         $OUT[1167] = ($FLAG[330] OR $FLAG[331] OR NOT $FLAG[330] AND NOT $FLAG[331] AND NOT $FLAG[332]) AND NOT $TIMER_FLAG[9]
      ;ENDFOLD
      ;FOLD -- Warte Fraesen fertig oder Timeout -- ;%{SE}%MKUKATPVW %CVW_COM %VCOMMENT %P 2:-- Warte Fraesen fertig oder Timeout --, 3: VW_COMMENT
      ;ENDFOLD
      ;FOLD Schritt 107 = (F175 & F190 + F174 & F186 & !F287 + T7 + T9 + F325) & A4039  ;%{SE}%MKUKATPVW %CVW_SPS %VST_CON %P 2:Schritt 107 = (F175 & F190 + F174 & F186 & !F287 + T7 + T9 + F325) & A4039 , 3: ST_CON
         IF ($FLAG[175] AND $FLAG[190] OR $FLAG[174] AND $FLAG[186] AND NOT $FLAG[287] OR $TIMER_FLAG[7] OR $TIMER_FLAG[9] OR $FLAG[325]) AND $OUT[4039] THEN
            PREVSTEP = $APP_INT[5]
            $APP_INT[5] = 107
         ENDIF
      ;ENDFOLD
      ;FOLD Schritt 107 = (F174 & F188 & F287 + T7 + T9 + F325) & A4039  ;%{SE}%MKUKATPVW %CVW_SPS %VST_CON %P 2:Schritt 107 = (F174 & F188 & F287 + T7 + T9 + F325) & A4039 , 3: ST_CON
         IF ($FLAG[174] AND $FLAG[188] AND $FLAG[287] OR $TIMER_FLAG[7] OR $TIMER_FLAG[9] OR $FLAG[325]) AND $OUT[4039] THEN
            PREVSTEP = $APP_INT[5]
            $APP_INT[5] = 107
         ENDIF
      ;ENDFOLD
   ;ENDFOLD
   ;FOLD SCHRITT 107 -- STAT EZ3/SP3/KE3 -- ;%{P}%MKUKATPVW,%CSTEP,%VST_NR,%P 1:SCHRITT, 2:107, 3: STAT EZ3/SP3/KE3
      ;FOLD ;%{H}
         Case 107
      ;ENDFOLD
      ;FOLD t9 ( EIN ) = STOP ;%{SE}%MKUKATPVW %CVW_SPS %VTSTOP %P 2:t9 ( EIN ) = STOP, 3: TSTOP
         VW(#SET_TIME,TRUE,9,1,0)
      ;ENDFOLD
      ;FOLD -- EZ3/SP3/KE3 oeffnen -- ;%{SE}%MKUKATPVW %CVW_COM %VCOMMENT %P 2:-- EZ3/SP3/KE3 oeffnen --, 3: VW_COMMENT
      ;ENDFOLD
      ;FOLD A1039 = AUS ;%{SE}%MKUKATPVW %CVW_SPS %VBOASG %P 2:A1039 = AUS, 3: BOASG
         $OUT[1039] = FALSE
      ;ENDFOLD
      ;FOLD A1038 = AUS ;%{SE}%MKUKATPVW %CVW_SPS %VBOASG %P 2:A1038 = AUS, 3: BOASG
         $OUT[1038] = FALSE
      ;ENDFOLD
      ;FOLD A1037 = EIN ;%{SE}%MKUKATPVW %CVW_SPS %VBOASG %P 2:A1037 = EIN, 3: BOASG
         $OUT[1037] = TRUE
      ;ENDFOLD
      ;FOLD -- KF3 Ausblasen -- ;%{SE}%MKUKATPVW %CVW_COM %VCOMMENT %P 2:-- KF3 Ausblasen --, 3: VW_COMMENT
      ;ENDFOLD
      ;FOLD A1167 = F330 + F331 + F332 + !F330 & !F331 & !F332 ;%{SE}%MKUKATPVW %CVW_SPS %VBOASG %P 2:A1167 = F330 + F331 + F332 + !F330 & !F331 & !F332, 3: BOASG
         $OUT[1167] = $FLAG[330] OR $FLAG[331] OR $FLAG[332] OR NOT $FLAG[330] AND NOT $FLAG[331] AND NOT $FLAG[332]
      ;ENDFOLD
      ;FOLD -- KF Ausblasen Ausschaltverzoegerung starten -- ;%{SE}%MKUKATPVW %CVW_COM %VCOMMENT %P 2:-- KF Ausblasen Ausschaltverzoegerung starten --, 3: VW_COMMENT
      ;ENDFOLD
      ;FOLD F739 = EIN ;%{SE}%MKUKATPVW %CVW_SPS %VBOASG %P 2:F739 = EIN, 3: BOASG
         $FLAG[739] = TRUE
      ;ENDFOLD
      ;FOLD -- RSK Sammelstoerung -- ;%{SE}%MKUKATPVW %CVW_COM %VCOMMENT %P 2:-- RSK Sammelstoerung --, 3: VW_COMMENT
      ;ENDFOLD
      ;FOLD F329 = T7 + T9 + F325 ;%{SE}%MKUKATPVW %CVW_SPS %VBOASG %P 2:F329 = T7 + T9 + F325, 3: BOASG
         $FLAG[329] = $TIMER_FLAG[7] OR $TIMER_FLAG[9] OR $FLAG[325]
      ;ENDFOLD
      ;FOLD -- Hilfsflag Startfraesen -- ;%{SE}%MKUKATPVW %CVW_COM %VCOMMENT %P 2:-- Hilfsflag Startfraesen --, 3: VW_COMMENT
      ;ENDFOLD
      ;FOLD F188 = (F188 & F174 + F190 & F175) & F287 ;%{SE}%MKUKATPVW %CVW_SPS %VBOASG %P 2:F188 = (F188 & F174 + F190 & F175) & F287, 3: BOASG
         $FLAG[188] = ($FLAG[188] AND $FLAG[174] OR $FLAG[190] AND $FLAG[175]) AND $FLAG[287]
      ;ENDFOLD
      ;FOLD F190 = !F200 & F190 + F200 & F287 & F190 ;%{SE}%MKUKATPVW %CVW_SPS %VBOASG %P 2:F190 = !F200 & F190 + F200 & F287 & F190, 3: BOASG
         $FLAG[190] = NOT $FLAG[200] AND $FLAG[190] OR $FLAG[200] AND $FLAG[287] AND $FLAG[190]
      ;ENDFOLD
      ;FOLD F287 = F174 + F175 & F200 ;%{SE}%MKUKATPVW %CVW_SPS %VBOASG %P 2:F287 = F174 + F175 & F200, 3: BOASG
         $FLAG[287] = $FLAG[174] OR $FLAG[175] AND $FLAG[200]
      ;ENDFOLD
      ;FOLD -- Neues Fraesprogramm und Zaehler ruecksetzen -- ;%{SE}%MKUKATPVW %CVW_COM %VCOMMENT %P 2:-- Neues Fraesprogramm und Zaehler ruecksetzen --, 3: VW_COMMENT
      ;ENDFOLD
      ;FOLD F270 = F188 & F732 ;%{SE}%MKUKATPVW %CVW_SPS %VBOASG %P 2:F270 = F188 & F732, 3: BOASG
         $FLAG[270] = $FLAG[188] AND $FLAG[732]
      ;ENDFOLD
      ;FOLD bin9 ( F732 ) = 36 ;%{SE}%MKUKATPVW %CVW_SPS %VARIASG %P 2:bin9 ( F732 ) = 36, 3: ARIASG
         VW(#BINOUT,$FLAG[732],9,36)
      ;ENDFOLD
      ;FOLD i19 ( F270 ) = i45 ;%{SE}%MKUKATPVW %CVW_SPS %VARIASG %P 2:i19 ( F270 ) = i45, 3: ARIASG
         VW(#COUNTER,$FLAG[270],19,$COUNT_I[45])
      ;ENDFOLD
      ;FOLD -- Wiederholung beim Startfraesen -- ;%{SE}%MKUKATPVW %CVW_COM %VCOMMENT %P 2:-- Wiederholung beim Startfraesen --, 3: VW_COMMENT
      ;ENDFOLD
      ;FOLD Schritt 104 = E1037 & !E1038 & (F174 & !F188 + F175 & F200 & !F188) & !F325 & !F329 & A4039  ;%{SE}%MKUKATPVW %CVW_SPS %VST_CON %P 2:Schritt 104 = E1037 & !E1038 & (F174 & !F188 + F175 & F200 & !F188) & !F325 & !F329 & A4039 , 3: ST_CON
         IF $IN[1037] AND NOT $IN[1038] AND ($FLAG[174] AND NOT $FLAG[188] OR $FLAG[175] AND $FLAG[200] AND NOT $FLAG[188]) AND NOT $FLAG[325] AND NOT $FLAG[329] AND $OUT[4039] THEN
            PREVSTEP = $APP_INT[5]
            $APP_INT[5] = 104
         ENDIF
      ;ENDFOLD
      ;FOLD -- Weiter wenn Fraesen fertig -- ;%{SE}%MKUKATPVW %CVW_COM %VCOMMENT %P 2:-- Weiter wenn Fraesen fertig --, 3: VW_COMMENT
      ;ENDFOLD
      ;FOLD Schritt 108 = E1037 & !E1038 & (F175 & F190 & (!F200 + F188)+ F174 & F188 + F325 + F329) & A4039  ;%{SE}%MKUKATPVW %CVW_SPS %VST_CON %P 2:Schritt 108 = E1037 & !E1038 & (F175 & F190 & (!F200 + F188)+ F174 & F188 + F325 + F329) & A4039 , 3: ST_CON
         IF $IN[1037] AND NOT $IN[1038] AND ($FLAG[175] AND $FLAG[190] AND (NOT $FLAG[200] OR $FLAG[188]) OR $FLAG[174] AND $FLAG[188] OR $FLAG[325] OR $FLAG[329]) AND $OUT[4039] THEN
            PREVSTEP = $APP_INT[5]
            $APP_INT[5] = 108
         ENDIF
      ;ENDFOLD
   ;ENDFOLD
   ;FOLD SCHRITT 108 -- STAT EZ3/SP3/KE3 -- ;%{P}%MKUKATPVW,%CSTEP,%VST_NR,%P 1:SCHRITT, 2:108, 3: STAT EZ3/SP3/KE3
      ;FOLD ;%{H}
         Case 108
      ;ENDFOLD
      ;FOLD F270 = AUS ;%{SE}%MKUKATPVW %CVW_SPS %VBOASG %P 2:F270 = AUS, 3: BOASG
         $FLAG[270] = FALSE
      ;ENDFOLD
      ;FOLD F324 = AUS ;%{SE}%MKUKATPVW %CVW_SPS %VBOASG %P 2:F324 = AUS, 3: BOASG
         $FLAG[324] = FALSE
      ;ENDFOLD
      ;FOLD A1037 = AUS ;%{SE}%MKUKATPVW %CVW_SPS %VBOASG %P 2:A1037 = AUS, 3: BOASG
         $OUT[1037] = FALSE
      ;ENDFOLD
      ;FOLD -- KF3 abschalten -- ;%{SE}%MKUKATPVW %CVW_COM %VCOMMENT %P 2:-- KF3 abschalten --, 3: VW_COMMENT
      ;ENDFOLD
      ;FOLD A1154 = AUS ;%{SE}%MKUKATPVW %CVW_SPS %VBOASG %P 2:A1154 = AUS, 3: BOASG
         $OUT[1154] = FALSE
      ;ENDFOLD
      ;FOLD -- Ueberwachungszeit KF1 Versetzeinheit -- ;%{SE}%MKUKATPVW %CVW_COM %VCOMMENT %P 2:-- Ueberwachungszeit KF1 Versetzeinheit --, 3: VW_COMMENT
      ;ENDFOLD
      ;FOLD t8 ( EIN ) = -20[1/10Sek] ;%{SE}%MKUKATPVW %CVW_SPS %VTASG %P 2:t8 ( EIN ) = -20[1/10Sek], 3: TASG
         VW(#SET_TIME,TRUE,8,0,-20)
      ;ENDFOLD
      ;FOLD Schritt 109 = A4039  ;%{SE}%MKUKATPVW %CVW_SPS %VST_CON %P 2:Schritt 109 = A4039 , 3: ST_CON
         IF $OUT[4039] THEN
            PREVSTEP = $APP_INT[5]
            $APP_INT[5] = 109
         ENDIF
      ;ENDFOLD
   ;ENDFOLD
   ;FOLD SCHRITT 109 -- STAT EZ3/SP3/KE3-- ;%{P}%MKUKATPVW,%CSTEP,%VST_NR,%P 1:SCHRITT, 2:109, 3: STAT EZ3/SP3/KE3
      ;FOLD ;%{H}
         Case 109
      ;ENDFOLD
      ;FOLD F328 = AUS ;%{SE}%MKUKATPVW %CVW_SPS %VBOASG %P 2:F328 = AUS, 3: BOASG
         $FLAG[328] = FALSE
      ;ENDFOLD
      ;FOLD -- KF3 Versetzeinheit vor -- ;%{SE}%MKUKATPVW %CVW_COM %VCOMMENT %P 2:-- KF3 Versetzeinheit vor --, 3: VW_COMMENT
      ;ENDFOLD
      ;FOLD A1155 = F564 ;%{SE}%MKUKATPVW %CVW_SPS %VBOASG %P 2:A1155 = F564, 3: BOASG
         $OUT[1155] = $FLAG[564]
      ;ENDFOLD
      ;FOLD -- RSK Fehlerausgabe KS3 Arbeitsst. -- ;%{SE}%MKUKATPVW %CVW_COM %VCOMMENT %P 2:-- RSK Fehlerausgabe KS3 Arbeitsst. --, 3: VW_COMMENT
      ;ENDFOLD
      ;FOLD F324 = (E1162 + !E1163 + !E1164 + E1165) & !F323 & !F328 + F324 ;%{SE}%MKUKATPVW %CVW_SPS %VBOASG %P 2:F324 = (E1162 + !E1163 + !E1164 + E1165) & !F323 & !F328 + F324, 3: BOASG
         $FLAG[324] = ($IN[1162] OR NOT $IN[1163] OR NOT $IN[1164] OR $IN[1165]) AND NOT $FLAG[323] AND NOT $FLAG[328] OR $FLAG[324]
      ;ENDFOLD
      ;FOLD -- RSK Sammelstoerung -- ;%{SE}%MKUKATPVW %CVW_COM %VCOMMENT %P 2:-- RSK Sammelstoerung --, 3: VW_COMMENT
      ;ENDFOLD
      ;FOLD F329 = F324 + F325 ;%{SE}%MKUKATPVW %CVW_SPS %VBOASG %P 2:F329 = F324 + F325, 3: BOASG
         $FLAG[329] = $FLAG[324] OR $FLAG[325]
      ;ENDFOLD
      ;FOLD -- Ueberwachungszeit KS3 schwenken -- ;%{SE}%MKUKATPVW %CVW_COM %VCOMMENT %P 2:-- Ueberwachungszeit KS3 schwenken --, 3: VW_COMMENT
      ;ENDFOLD
      ;FOLD t9 ( EIN ) = -100[1/10Sek] ;%{SE}%MKUKATPVW %CVW_SPS %VTASG %P 2:t9 ( EIN ) = -100[1/10Sek], 3: TASG
         VW(#SET_TIME,TRUE,9,0,-100)
      ;ENDFOLD
      ;FOLD Schritt 108 = F324 & (E26 + E27) & A4039  ;%{SE}%MKUKATPVW %CVW_SPS %VST_CON %P 2:Schritt 108 = F324 & (E26 + E27) & A4039 , 3: ST_CON
         IF $FLAG[324] AND ($IN[26] OR $IN[27]) AND $OUT[4039] THEN
            PREVSTEP = $APP_INT[5]
            $APP_INT[5] = 108
         ENDIF
      ;ENDFOLD
      ;FOLD Schritt 110 = (!F324 & (E1155 & F564 + !E1155 & !F564) + T8 + F325) & A4039  ;%{SE}%MKUKATPVW %CVW_SPS %VST_CON %P 2:Schritt 110 = (!F324 & (E1155 & F564 + !E1155 & !F564) + T8 + F325) & A4039 , 3: ST_CON
         IF (NOT $FLAG[324] AND ($IN[1155] AND $FLAG[564] OR NOT $IN[1155] AND NOT $FLAG[564]) OR $TIMER_FLAG[8] OR $FLAG[325]) AND $OUT[4039] THEN
            PREVSTEP = $APP_INT[5]
            $APP_INT[5] = 110
         ENDIF
      ;ENDFOLD
   ;ENDFOLD
   ;FOLD SCHRITT 110 -- STAT EZ3/SP3/KE3-- ;%{P}%MKUKATPVW,%CSTEP,%VST_NR,%P 1:SCHRITT, 2:110, 3: STAT EZ3/SP3/KE3
      ;FOLD ;%{H}
         Case 110
      ;ENDFOLD
      ;FOLD F323 = AUS ;%{SE}%MKUKATPVW %CVW_SPS %VBOASG %P 2:F323 = AUS, 3: BOASG
         $FLAG[323] = FALSE
      ;ENDFOLD
      ;FOLD F328 = AUS ;%{SE}%MKUKATPVW %CVW_SPS %VBOASG %P 2:F328 = AUS, 3: BOASG
         $FLAG[328] = FALSE
      ;ENDFOLD
      ;FOLD -- RSK Sammelstoerung -- ;%{SE}%MKUKATPVW %CVW_COM %VCOMMENT %P 2:-- RSK Sammelstoerung --, 3: VW_COMMENT
      ;ENDFOLD
      ;FOLD F329 = F325 ;%{SE}%MKUKATPVW %CVW_SPS %VBOASG %P 2:F329 = F325, 3: BOASG
         $FLAG[329] = $FLAG[325]
      ;ENDFOLD
      ;FOLD -- KF3 ein -- ;%{SE}%MKUKATPVW %CVW_COM %VCOMMENT %P 2:-- KF3 ein --, 3: VW_COMMENT
      ;ENDFOLD
      ;FOLD A1154 = EIN ;%{SE}%MKUKATPVW %CVW_SPS %VBOASG %P 2:A1154 = EIN, 3: BOASG
         $OUT[1154] = TRUE
      ;ENDFOLD
      ;FOLD -- KS3 in Ruhestellung schwenken -- ;%{SE}%MKUKATPVW %CVW_COM %VCOMMENT %P 2:-- KS3 in Ruhestellung schwenken --, 3: VW_COMMENT
      ;ENDFOLD
      ;FOLD A1162 = (F747 + !F714) & (E1037 + F714) & (E1155 & F564 + !E1155 & !F564) ;%{SE}%MKUKATPVW %CVW_SPS %VBOASG %P 2:A1162 = (F747 + !F714) & (E1037 + F714) & (E1155 & F564 + !E1155 & !F564), 3: BOASG
         $OUT[1162] = ($FLAG[747] OR NOT $FLAG[714]) AND ($IN[1037] OR $FLAG[714]) AND ($IN[1155] AND $FLAG[564] OR NOT $IN[1155] AND NOT $FLAG[564])
      ;ENDFOLD
      ;FOLD Schritt 111 = (F747 + !F714 + T9) & (A1162 + T9) & (E1037 + F714) & A4039  ;%{SE}%MKUKATPVW %CVW_SPS %VST_CON %P 2:Schritt 111 = (F747 + !F714 + T9) & (A1162 + T9) & (E1037 + F714) & A4039 , 3: ST_CON
         IF ($FLAG[747] OR NOT $FLAG[714] OR $TIMER_FLAG[9]) AND ($OUT[1162] OR $TIMER_FLAG[9]) AND ($IN[1037] OR $FLAG[714]) AND $OUT[4039] THEN
            PREVSTEP = $APP_INT[5]
            $APP_INT[5] = 111
         ENDIF
      ;ENDFOLD
   ;ENDFOLD
   ;FOLD SCHRITT 111 -- STAT EZ3/SP3/KE3 -- ;%{P}%MKUKATPVW,%CSTEP,%VST_NR,%P 1:SCHRITT, 2:111, 3: STAT EZ3/SP3/KE3
      ;FOLD ;%{H}
         Case 111
      ;ENDFOLD
      ;FOLD -- Hilfsflag SK Programmwechsel -- ;%{SE}%MKUKATPVW %CVW_COM %VCOMMENT %P 2:-- Hilfsflag SK Programmwechsel --, 3: VW_COMMENT
      ;ENDFOLD
      ;FOLD F334 = AUS ;%{SE}%MKUKATPVW %CVW_SPS %VBOASG %P 2:F334 = AUS, 3: BOASG
         $FLAG[334] = FALSE
      ;ENDFOLD
      ;FOLD -- RSK Fehlerausgabe KF Versetzeinheit -- ;%{SE}%MKUKATPVW %CVW_COM %VCOMMENT %P 2:-- RSK Fehlerausgabe KF Versetzeinheit --, 3: VW_COMMENT
      ;ENDFOLD
      ;FOLD F328 = !E1155 & F564 & !F323 + F328 ;%{SE}%MKUKATPVW %CVW_SPS %VBOASG %P 2:F328 = !E1155 & F564 & !F323 + F328, 3: BOASG
         $FLAG[328] = NOT $IN[1155] AND $FLAG[564] AND NOT $FLAG[323] OR $FLAG[328]
      ;ENDFOLD
      ;FOLD -- RSK Fehlerausgabe KS3 Ruhestellung -- ;%{SE}%MKUKATPVW %CVW_COM %VCOMMENT %P 2:-- RSK Fehlerausgabe KS3 Ruhestellung --, 3: VW_COMMENT
      ;ENDFOLD
      ;FOLD F323 = (!E1162 + E1163 + E1164 + !E1165) & T9 & (E1155 + !F564) + F323 ;%{SE}%MKUKATPVW %CVW_SPS %VBOASG %P 2:F323 = (!E1162 + E1163 + E1164 + !E1165) & T9 & (E1155 + !F564) + F323, 3: BOASG
         $FLAG[323] = (NOT $IN[1162] OR $IN[1163] OR $IN[1164] OR NOT $IN[1165]) AND $TIMER_FLAG[9] AND ($IN[1155] OR NOT $FLAG[564]) OR $FLAG[323]
      ;ENDFOLD
      ;FOLD -- RSK Fehlerausgabe EZ/SP min. Oeffnung -- ;%{SE}%MKUKATPVW %CVW_COM %VCOMMENT %P 2:-- RSK Fehlerausgabe EZ/SP min. Oeffnung --, 3: VW_COMMENT
      ;ENDFOLD
      ;FOLD F333 = !F747 ;%{SE}%MKUKATPVW %CVW_SPS %VBOASG %P 2:F333 = !F747, 3: BOASG
         $FLAG[333] = NOT $FLAG[747]
      ;ENDFOLD
      ;FOLD -- RSK Sammelstoerung -- ;%{SE}%MKUKATPVW %CVW_COM %VCOMMENT %P 2:-- RSK Sammelstoerung --, 3: VW_COMMENT
      ;ENDFOLD
      ;FOLD F329 = F323 + F325 + F328 ;%{SE}%MKUKATPVW %CVW_SPS %VBOASG %P 2:F329 = F323 + F325 + F328, 3: BOASG
         $FLAG[329] = $FLAG[323] OR $FLAG[325] OR $FLAG[328]
      ;ENDFOLD
      ;FOLD A1154 = !F323 & !F328 ;%{SE}%MKUKATPVW %CVW_SPS %VBOASG %P 2:A1154 = !F323 & !F328, 3: BOASG
         $OUT[1154] = NOT $FLAG[323] AND NOT $FLAG[328]
      ;ENDFOLD
      ;FOLD A1155 = F564 ;%{SE}%MKUKATPVW %CVW_SPS %VBOASG %P 2:A1155 = F564, 3: BOASG
         $OUT[1155] = $FLAG[564]
      ;ENDFOLD
      ;FOLD Schritt 109 = (F323 + F328) & (E26 + E27) & A4039  ;%{SE}%MKUKATPVW %CVW_SPS %VST_CON %P 2:Schritt 109 = (F323 + F328) & (E26 + E27) & A4039 , 3: ST_CON
         IF ($FLAG[323] OR $FLAG[328]) AND ($IN[26] OR $IN[27]) AND $OUT[4039] THEN
            PREVSTEP = $APP_INT[5]
            $APP_INT[5] = 109
         ENDIF
      ;ENDFOLD
      ;FOLD Schritt 112 = !A1162 & E1162 & !E1163 & !E1164 & E1165 & A4039  ;%{SE}%MKUKATPVW %CVW_SPS %VST_CON %P 2:Schritt 112 = !A1162 & E1162 & !E1163 & !E1164 & E1165 & A4039 , 3: ST_CON
         IF NOT $OUT[1162] AND $IN[1162] AND NOT $IN[1163] AND NOT $IN[1164] AND $IN[1165] AND $OUT[4039] THEN
            PREVSTEP = $APP_INT[5]
            $APP_INT[5] = 112
         ENDIF
      ;ENDFOLD
   ;ENDFOLD
   ;FOLD SCHRITT 112 -- STAT EZ3/SP3/KE3-- ;%{P}%MKUKATPVW,%CSTEP,%VST_NR,%P 1:SCHRITT, 2:112, 3: STAT EZ3/SP3/KE3
      ;FOLD ;%{H}
         Case 112
      ;ENDFOLD
      ;FOLD F323 = AUS ;%{SE}%MKUKATPVW %CVW_SPS %VBOASG %P 2:F323 = AUS, 3: BOASG
         $FLAG[323] = FALSE
      ;ENDFOLD
      ;FOLD F328 = AUS ;%{SE}%MKUKATPVW %CVW_SPS %VBOASG %P 2:F328 = AUS, 3: BOASG
         $FLAG[328] = FALSE
      ;ENDFOLD
      ;FOLD -- RSK Sammelstoerung -- ;%{SE}%MKUKATPVW %CVW_COM %VCOMMENT %P 2:-- RSK Sammelstoerung --, 3: VW_COMMENT
      ;ENDFOLD
      ;FOLD F329 = F325 ;%{SE}%MKUKATPVW %CVW_SPS %VBOASG %P 2:F329 = F325, 3: BOASG
         $FLAG[329] = $FLAG[325]
      ;ENDFOLD
      ;FOLD t9 ( EIN ) = STOP ;%{SE}%MKUKATPVW %CVW_SPS %VTSTOP %P 2:t9 ( EIN ) = STOP, 3: TSTOP
         VW(#SET_TIME,TRUE,9,1,0)
      ;ENDFOLD
      ;FOLD -- KF1 Versetzeinheit rueck -- ;%{SE}%MKUKATPVW %CVW_COM %VCOMMENT %P 2:-- KF1 Versetzeinheit rueck --, 3: VW_COMMENT
      ;ENDFOLD
      ;FOLD A1155 = AUS ;%{SE}%MKUKATPVW %CVW_SPS %VBOASG %P 2:A1155 = AUS, 3: BOASG
         $OUT[1155] = FALSE
      ;ENDFOLD
      ;FOLD -- KF3 aus -- ;%{SE}%MKUKATPVW %CVW_COM %VCOMMENT %P 2:-- KF3 aus --, 3: VW_COMMENT
      ;ENDFOLD
      ;FOLD A1154 = AUS ;%{SE}%MKUKATPVW %CVW_SPS %VBOASG %P 2:A1154 = AUS, 3: BOASG
         $OUT[1154] = FALSE
      ;ENDFOLD
      ;FOLD -- KF1 Ausblasen -- ;%{SE}%MKUKATPVW %CVW_COM %VCOMMENT %P 2:-- KF1 Ausblasen --, 3: VW_COMMENT
      ;ENDFOLD
      ;FOLD A1167 = (F330 + F331 + F332) & F739 ;%{SE}%MKUKATPVW %CVW_SPS %VBOASG %P 2:A1167 = (F330 + F331 + F332) & F739, 3: BOASG
         $OUT[1167] = ($FLAG[330] OR $FLAG[331] OR $FLAG[332]) AND $FLAG[739]
      ;ENDFOLD
      ;FOLD bin9 ( !F329 ) = 1 ;%{SE}%MKUKATPVW %CVW_SPS %VARIASG %P 2:bin9 ( !F329 ) = 1, 3: ARIASG
         VW(#BINOUT,NOT $FLAG[329],9,1)
      ;ENDFOLD
      ;FOLD -- Wartezeit Programmwechsel SK -- ;%{SE}%MKUKATPVW %CVW_COM %VCOMMENT %P 2:-- Wartezeit Programmwechsel SK --, 3: VW_COMMENT
      ;ENDFOLD
      ;FOLD t8 ( !F334 ) = -2[1/10Sek] ;%{SE}%MKUKATPVW %CVW_SPS %VTASG %P 2:t8 ( !F334 ) = -2[1/10Sek], 3: TASG
         VW(#SET_TIME,NOT $FLAG[334],8,0,-2)
      ;ENDFOLD
      ;FOLD -- Hilfsflag SK Programmwechsel -- ;%{SE}%MKUKATPVW %CVW_COM %VCOMMENT %P 2:-- Hilfsflag SK Programmwechsel --, 3: VW_COMMENT
      ;ENDFOLD
      ;FOLD F334 = EIN ;%{SE}%MKUKATPVW %CVW_SPS %VBOASG %P 2:F334 = EIN, 3: BOASG
         $FLAG[334] = TRUE
      ;ENDFOLD
      ;FOLD -- Ueberwachungszeit EZ3/SP3/KE3 Messen -- ;%{SE}%MKUKATPVW %CVW_COM %VCOMMENT %P 2:-- Ueberwachungszeit EZ3/SP3/KE3 Messen --, 3: VW_COMMENT
      ;ENDFOLD
      ;FOLD t9 ( EIN ) = -150[1/10Sek] ;%{SE}%MKUKATPVW %CVW_SPS %VTASG %P 2:t9 ( EIN ) = -150[1/10Sek], 3: TASG
         VW(#SET_TIME,TRUE,9,0,-150)
      ;ENDFOLD
      ;FOLD Schritt 97 = (F325 + F329) & (E26 + E27) & A4039  ;%{SE}%MKUKATPVW %CVW_SPS %VST_CON %P 2:Schritt 97 = (F325 + F329) & (E26 + E27) & A4039 , 3: ST_CON
         IF ($FLAG[325] OR $FLAG[329]) AND ($IN[26] OR $IN[27]) AND $OUT[4039] THEN
            PREVSTEP = $APP_INT[5]
            $APP_INT[5] = 97
         ENDIF
      ;ENDFOLD
      ;FOLD Schritt 113 = T8 & !F325 & !F329 & A4039  ;%{SE}%MKUKATPVW %CVW_SPS %VST_CON %P 2:Schritt 113 = T8 & !F325 & !F329 & A4039 , 3: ST_CON
         IF $TIMER_FLAG[8] AND NOT $FLAG[325] AND NOT $FLAG[329] AND $OUT[4039] THEN
            PREVSTEP = $APP_INT[5]
            $APP_INT[5] = 113
         ENDIF
      ;ENDFOLD
   ;ENDFOLD
   ;FOLD SCHRITT 113 -- STAT EZ3/SP3/KE3 -- ;%{P}%MKUKATPVW,%CSTEP,%VST_NR,%P 1:SCHRITT, 2:113, 3: STAT EZ3/SP3/KE3
      ;FOLD ;%{H}
         Case 113
      ;ENDFOLD
      ;FOLD -- Hilfsflag SK Programmwechsel -- ;%{SE}%MKUKATPVW %CVW_COM %VCOMMENT %P 2:-- Hilfsflag SK Programmwechsel --, 3: VW_COMMENT
      ;ENDFOLD
      ;FOLD F334 = AUS ;%{SE}%MKUKATPVW %CVW_SPS %VBOASG %P 2:F334 = AUS, 3: BOASG
         $FLAG[334] = FALSE
      ;ENDFOLD
      ;FOLD -- Quitt. Fraesen SK3 -- ;%{SE}%MKUKATPVW %CVW_COM %VCOMMENT %P 2:-- Quitt. Fraesen SK3 --, 3: VW_COMMENT
      ;ENDFOLD
      ;FOLD A1106 = (!F329 & !F322 & !F832) + ( F832 & A1106) ;%{SE}%MKUKATPVW %CVW_SPS %VBOASG %P 2:A1106 = (!F329 & !F322 & !F832) + ( F832 & A1106), 3: BOASG
         $OUT[1106] = (NOT $FLAG[329] AND NOT $FLAG[322] AND NOT $FLAG[832]) OR ($FLAG[832] AND $OUT[1106])
      ;ENDFOLD
      ;FOLD A1042 = (!F329 & !F322 & F832) + ( !F832 & A1042) ;%{SE}%MKUKATPVW %CVW_SPS %VBOASG %P 2:A1042 = (!F329 & !F322 & F832) + ( !F832 & A1042), 3: BOASG
         $OUT[1042] = (NOT $FLAG[329] AND NOT $FLAG[322] AND $FLAG[832]) OR (NOT $FLAG[832] AND $OUT[1042])
      ;ENDFOLD
      ;FOLD -- RSK Sammelstoerung -- ;%{SE}%MKUKATPVW %CVW_COM %VCOMMENT %P 2:-- RSK Sammelstoerung --, 3: VW_COMMENT
      ;ENDFOLD
      ;FOLD F329 = T9 ;%{SE}%MKUKATPVW %CVW_SPS %VBOASG %P 2:F329 = T9, 3: BOASG
         $FLAG[329] = $TIMER_FLAG[9]
      ;ENDFOLD
      ;FOLD -- Messen nach Fraesen -- ;%{SE}%MKUKATPVW %CVW_COM %VCOMMENT %P 2:-- Messen nach Fraesen --, 3: VW_COMMENT
      ;ENDFOLD
      ;FOLD A1079 = (!F174 & F175 & !F832) + (F832 & A1079) ;%{SE}%MKUKATPVW %CVW_SPS %VBOASG %P 2:A1079 = (!F174 & F175 & !F832) + (F832 & A1079), 3: BOASG
         $OUT[1079] = (NOT $FLAG[174] AND $FLAG[175] AND NOT $FLAG[832]) OR ($FLAG[832] AND $OUT[1079])
      ;ENDFOLD
      ;FOLD A1078 = (F174 & !F175 & !F832) + (F832 & A1078) ;%{SE}%MKUKATPVW %CVW_SPS %VBOASG %P 2:A1078 = (F174 & !F175 & !F832) + (F832 & A1078), 3: BOASG
         $OUT[1078] = ($FLAG[174] AND NOT $FLAG[175] AND NOT $FLAG[832]) OR ($FLAG[832] AND $OUT[1078])
      ;ENDFOLD
      ;FOLD F836 = (F174 + F175) & !F329 ;%{SE}%MKUKATPVW %CVW_SPS %VBOASG %P 2:F836 = (F174 + F175) & !F329, 3: BOASG
         $FLAG[836] = ($FLAG[174] OR $FLAG[175]) AND NOT $FLAG[329]
      ;ENDFOLD
      ;FOLD A1077 = (F836 & !F832) + (F832 & A1077) ;%{SE}%MKUKATPVW %CVW_SPS %VBOASG %P 2:A1077 = (F836 & !F832) + (F832 & A1077), 3: BOASG
         $OUT[1077] = ($FLAG[836] AND NOT $FLAG[832]) OR ($FLAG[832] AND $OUT[1077])
      ;ENDFOLD
      ;FOLD A1045 = (F836 & F832) + (!F832 & A1045) ;%{SE}%MKUKATPVW %CVW_SPS %VBOASG %P 2:A1045 = (F836 & F832) + (!F832 & A1045), 3: BOASG
         $OUT[1045] = ($FLAG[836] AND $FLAG[832]) OR (NOT $FLAG[832] AND $OUT[1045])
      ;ENDFOLD
      ;FOLD Schritt 114 = !E1106 & E1107 & !E1108 & A4039  ;%{SE}%MKUKATPVW %CVW_SPS %VST_CON %P 2:Schritt 114 = !E1106 & E1107 & !E1108 & A4039 , 3: ST_CON
         IF NOT $IN[1106] AND $IN[1107] AND NOT $IN[1108] AND $OUT[4039] THEN
            PREVSTEP = $APP_INT[5]
            $APP_INT[5] = 114
         ENDIF
      ;ENDFOLD
   ;ENDFOLD
   ;FOLD SCHRITT 114 -- STAT EZ3/SP3/KE3 -- ;%{P}%MKUKATPVW,%CSTEP,%VST_NR,%P 1:SCHRITT, 2:114, 3: STAT EZ3/SP3/KE3
      ;FOLD ;%{H}
         Case 114
      ;ENDFOLD
      ;FOLD -- Hilfsflag SK Programmwechsel -- ;%{SE}%MKUKATPVW %CVW_COM %VCOMMENT %P 2:-- Hilfsflag SK Programmwechsel --, 3: VW_COMMENT
      ;ENDFOLD
      ;FOLD F334 = AUS ;%{SE}%MKUKATPVW %CVW_SPS %VBOASG %P 2:F334 = AUS, 3: BOASG
         $FLAG[334] = FALSE
      ;ENDFOLD
      ;FOLD -- RSK Sammelstoerung -- ;%{SE}%MKUKATPVW %CVW_COM %VCOMMENT %P 2:-- RSK Sammelstoerung --, 3: VW_COMMENT
      ;ENDFOLD
      ;FOLD F329 = T9 ;%{SE}%MKUKATPVW %CVW_SPS %VBOASG %P 2:F329 = T9, 3: BOASG
         $FLAG[329] = $TIMER_FLAG[9]
      ;ENDFOLD
      ;FOLD Schritt 115 = A4039 & E1037 & (E1077 & !E1096 & !F832 + T9) + ( E1045 & !E1096 & F832 + T9)  ;%{SE}%MKUKATPVW %CVW_SPS %VST_CON %P 2:Schritt 115 = A4039 & E1037 & (E1077 & !E1096 & !F832 + T9) + ( E1045 & !E1096 & F832 + T9) , 3: ST_CON
         IF $OUT[4039] AND $IN[1037] AND ($IN[1077] AND NOT $IN[1096] AND NOT $FLAG[832] OR $TIMER_FLAG[9]) OR ($IN[1045] AND NOT $IN[1096] AND $FLAG[832] OR $TIMER_FLAG[9]) THEN
            PREVSTEP = $APP_INT[5]
            $APP_INT[5] = 115
         ENDIF
      ;ENDFOLD
   ;ENDFOLD
   ;FOLD SCHRITT 115 -- STAT EZ3/SP3/KE3 -- ;%{P}%MKUKATPVW,%CSTEP,%VST_NR,%P 1:SCHRITT, 2:115, 3: STAT EZ3/SP3/KE3
      ;FOLD ;%{H}
         Case 115
      ;ENDFOLD
      ;FOLD F836 = AUS ;%{SE}%MKUKATPVW %CVW_SPS %VBOASG %P 2:F836 = AUS, 3: BOASG
         $FLAG[836] = FALSE
      ;ENDFOLD
      ;FOLD t9 ( EIN ) = STOP ;%{SE}%MKUKATPVW %CVW_SPS %VTSTOP %P 2:t9 ( EIN ) = STOP, 3: TSTOP
         VW(#SET_TIME,TRUE,9,1,0)
      ;ENDFOLD
      ;FOLD -- RSK Fehlerausgabe Kappenverschleiss -- ;%{SE}%MKUKATPVW %CVW_COM %VCOMMENT %P 2:-- RSK Fehlerausgabe Kappenverschleiss --, 3: VW_COMMENT
      ;ENDFOLD
      ;FOLD F196 = E1097 ;%{SE}%MKUKATPVW %CVW_SPS %VBOASG %P 2:F196 = E1097, 3: BOASG
         $FLAG[196] = $IN[1097]
      ;ENDFOLD
      ;FOLD -- RSK Fehlerausgabe Messen -- ;%{SE}%MKUKATPVW %CVW_COM %VCOMMENT %P 2:-- RSK Fehlerausgabe Messen --, 3: VW_COMMENT
      ;ENDFOLD
      ;FOLD F326 = E1096 + E1097 + E1098 + F326 ;%{SE}%MKUKATPVW %CVW_SPS %VBOASG %P 2:F326 = E1096 + E1097 + E1098 + F326, 3: BOASG
         $FLAG[326] = $IN[1096] OR $IN[1097] OR $IN[1098] OR $FLAG[326]
      ;ENDFOLD
      ;FOLD -- RSK Sammelstoerung -- ;%{SE}%MKUKATPVW %CVW_COM %VCOMMENT %P 2:-- RSK Sammelstoerung --, 3: VW_COMMENT
      ;ENDFOLD
      ;FOLD F329 = F326 ;%{SE}%MKUKATPVW %CVW_SPS %VBOASG %P 2:F329 = F326, 3: BOASG
         $FLAG[329] = $FLAG[326]
      ;ENDFOLD
      ;FOLD A1078 = F832 & A1078 ;%{SE}%MKUKATPVW %CVW_SPS %VBOASG %P 2:A1078 = F832 & A1078, 3: BOASG
         $OUT[1078] = $FLAG[832] AND $OUT[1078]
      ;ENDFOLD
      ;FOLD A1079 = F832 & A1079 ;%{SE}%MKUKATPVW %CVW_SPS %VBOASG %P 2:A1079 = F832 & A1079, 3: BOASG
         $OUT[1079] = $FLAG[832] AND $OUT[1079]
      ;ENDFOLD
      ;FOLD -- Druckvorgabe SK3/EZ3/SP3/KE3 -- ;%{SE}%MKUKATPVW %CVW_COM %VCOMMENT %P 2:-- Druckvorgabe SK3/EZ3/SP3/KE3 --, 3: VW_COMMENT
      ;ENDFOLD
      ;FOLD bin7 ( F174 ) = 41 ;%{SE}%MKUKATPVW %CVW_SPS %VARIASG %P 2:bin7 ( F174 ) = 41, 3: ARIASG
         VW(#BINOUT,$FLAG[174],7,41)
      ;ENDFOLD
      ;FOLD bin7 ( F175 ) = 51 ;%{SE}%MKUKATPVW %CVW_SPS %VARIASG %P 2:bin7 ( F175 ) = 51, 3: ARIASG
         VW(#BINOUT,$FLAG[175],7,51)
      ;ENDFOLD
      ;FOLD bin9 ( F174 ) = 41 ;%{SE}%MKUKATPVW %CVW_SPS %VARIASG %P 2:bin9 ( F174 ) = 41, 3: ARIASG
         VW(#BINOUT,$FLAG[174],9,41)
      ;ENDFOLD
      ;FOLD bin9 ( F175 ) = 51 ;%{SE}%MKUKATPVW %CVW_SPS %VARIASG %P 2:bin9 ( F175 ) = 51, 3: ARIASG
         VW(#BINOUT,$FLAG[175],9,51)
      ;ENDFOLD
      ;FOLD -- Wartezeit Programmwechsel SK -- ;%{SE}%MKUKATPVW %CVW_COM %VCOMMENT %P 2:-- Wartezeit Programmwechsel SK --, 3: VW_COMMENT
      ;ENDFOLD
      ;FOLD T8 ( !F334 ) = -2[1/10Sek] ;%{SE}%MKUKATPVW %CVW_SPS %VTASG %P 2:T8 ( !F334 ) = -2[1/10Sek], 3: TASG
         VW(#SET_TIME,NOT $FLAG[334],8,0,-2)
      ;ENDFOLD
      ;FOLD -- Hilfsflag SK Programmwechsel -- ;%{SE}%MKUKATPVW %CVW_COM %VCOMMENT %P 2:-- Hilfsflag SK Programmwechsel --, 3: VW_COMMENT
      ;ENDFOLD
      ;FOLD F334 = EIN ;%{SE}%MKUKATPVW %CVW_SPS %VBOASG %P 2:F334 = EIN, 3: BOASG
         $FLAG[334] = TRUE
      ;ENDFOLD
      ;FOLD -- Ueberwachungszeit EZ3/SP3/KE3 Setzhub 2 -- ;%{SE}%MKUKATPVW %CVW_COM %VCOMMENT %P 2:-- Ueberwachungszeit EZ3/SP3/KE3 Setzhub 2 --, 3: VW_COMMENT
      ;ENDFOLD
      ;FOLD t9 ( EIN ) = -80[1/10Sek] ;%{SE}%MKUKATPVW %CVW_SPS %VTASG %P 2:t9 ( EIN ) = -80[1/10Sek], 3: TASG
         VW(#SET_TIME,TRUE,9,0,-80)
      ;ENDFOLD
      ;FOLD Schritt 116 = T8 & !F335 & A4039  ;%{SE}%MKUKATPVW %CVW_SPS %VST_CON %P 2:Schritt 116 = T8 & !F335 & A4039 , 3: ST_CON
         IF $TIMER_FLAG[8] AND NOT $FLAG[335] AND $OUT[4039] THEN
            PREVSTEP = $APP_INT[5]
            $APP_INT[5] = 116
         ENDIF
      ;ENDFOLD
      ;FOLD Schritt 116 = T8 & F335 & !F174 & A4039  ;%{SE}%MKUKATPVW %CVW_SPS %VST_CON %P 2:Schritt 116 = T8 & F335 & !F174 & A4039 , 3: ST_CON
         IF $TIMER_FLAG[8] AND $FLAG[335] AND NOT $FLAG[174] AND $OUT[4039] THEN
            PREVSTEP = $APP_INT[5]
            $APP_INT[5] = 116
         ENDIF
      ;ENDFOLD
      ;FOLD Schritt 227 = T8 & F335 & F174 & A4039  ;%{SE}%MKUKATPVW %CVW_SPS %VST_CON %P 2:Schritt 227 = T8 & F335 & F174 & A4039 , 3: ST_CON
         IF $TIMER_FLAG[8] AND $FLAG[335] AND $FLAG[174] AND $OUT[4039] THEN
            PREVSTEP = $APP_INT[5]
            $APP_INT[5] = 227
         ENDIF
      ;ENDFOLD
   ;ENDFOLD
   ;FOLD SCHRITT 116 -- STAT EZ3/SP3 -- ;%{P}%MKUKATPVW,%CSTEP,%VST_NR,%P 1:SCHRITT, 2:116, 3: STAT EZ3/SP3
      ;FOLD ;%{H}
         Case 116
      ;ENDFOLD
      ;FOLD -- Hilfsflag SK Programmwechsel -- ;%{SE}%MKUKATPVW %CVW_COM %VCOMMENT %P 2:-- Hilfsflag SK Programmwechsel --, 3: VW_COMMENT
      ;ENDFOLD
      ;FOLD F334 = AUS ;%{SE}%MKUKATPVW %CVW_SPS %VBOASG %P 2:F334 = AUS, 3: BOASG
         $FLAG[334] = FALSE
      ;ENDFOLD
      ;FOLD A1077 = F832 & A1077 ;%{SE}%MKUKATPVW %CVW_SPS %VBOASG %P 2:A1077 = F832 & A1077, 3: BOASG
         $OUT[1077] = $FLAG[832] AND $OUT[1077]
      ;ENDFOLD
      ;FOLD -- EZ3/SP3/KE3 schliessen -- ;%{SE}%MKUKATPVW %CVW_COM %VCOMMENT %P 2:-- EZ3/SP3/KE3 schliessen --, 3: VW_COMMENT
      ;ENDFOLD
      ;FOLD A1045 = !F832 & A1045 ;%{SE}%MKUKATPVW %CVW_SPS %VBOASG %P 2:A1045 = !F832 & A1045, 3: BOASG
         $OUT[1045] = NOT $FLAG[832] AND $OUT[1045]
      ;ENDFOLD
      ;FOLD A1037 = AUS ;%{SE}%MKUKATPVW %CVW_SPS %VBOASG %P 2:A1037 = AUS, 3: BOASG
         $OUT[1037] = FALSE
      ;ENDFOLD
      ;FOLD A1038 = !F329 & !F196 ;%{SE}%MKUKATPVW %CVW_SPS %VBOASG %P 2:A1038 = !F329 & !F196, 3: BOASG
         $OUT[1038] = NOT $FLAG[329] AND NOT $FLAG[196]
      ;ENDFOLD
      ;FOLD -- Ueberwachungszeit Kurzschlussschweissung SK3 -- ;%{SE}%MKUKATPVW %CVW_COM %VCOMMENT %P 2:-- Ueberwachungszeit Kurzschlussschweissung SK3 --, 3: VW_COMMENT
      ;ENDFOLD
      ;FOLD t9 ( EIN ) = -80[1/10Sek] ;%{SE}%MKUKATPVW %CVW_SPS %VTASG %P 2:t9 ( EIN ) = -80[1/10Sek], 3: TASG
         VW(#SET_TIME,TRUE,9,0,-80)
      ;ENDFOLD
      ;FOLD Schritt 117 = !E1037 & E1038 + E1037 & !E1038 & (F329 + F326 + F196) & A4039  ;%{SE}%MKUKATPVW %CVW_SPS %VST_CON %P 2:Schritt 117 = !E1037 & E1038 + E1037 & !E1038 & (F329 + F326 + F196) & A4039 , 3: ST_CON
         IF NOT $IN[1037] AND $IN[1038] OR $IN[1037] AND NOT $IN[1038] AND ($FLAG[329] OR $FLAG[326] OR $FLAG[196]) AND $OUT[4039] THEN
            PREVSTEP = $APP_INT[5]
            $APP_INT[5] = 117
         ENDIF
      ;ENDFOLD
   ;ENDFOLD
   ;FOLD SCHRITT 117 -- STAT EZ3/SP3/KE3-- ;%{P}%MKUKATPVW,%CSTEP,%VST_NR,%P 1:SCHRITT, 2:117, 3: STAT EZ3/SP3/KE3
      ;FOLD ;%{H}
         Case 117
      ;ENDFOLD
      ;FOLD -- Hilfsflag SK Programmwechsel -- ;%{SE}%MKUKATPVW %CVW_COM %VCOMMENT %P 2:-- Hilfsflag SK Programmwechsel --, 3: VW_COMMENT
      ;ENDFOLD
      ;FOLD F334 = AUS ;%{SE}%MKUKATPVW %CVW_SPS %VBOASG %P 2:F334 = AUS, 3: BOASG
         $FLAG[334] = FALSE
      ;ENDFOLD
      ;FOLD t9 ( EIN ) = STOP ;%{SE}%MKUKATPVW %CVW_SPS %VTSTOP %P 2:t9 ( EIN ) = STOP, 3: TSTOP
         VW(#SET_TIME,TRUE,9,1,0)
      ;ENDFOLD
      ;FOLD -- RSK Fehlerausgabe Kraftaufbau -- ;%{SE}%MKUKATPVW %CVW_COM %VCOMMENT %P 2:-- RSK Fehlerausgabe Kraftaufbau --, 3: VW_COMMENT
      ;ENDFOLD
      ;FOLD F325 = T9 + F325 ;%{SE}%MKUKATPVW %CVW_SPS %VBOASG %P 2:F325 = T9 + F325, 3: BOASG
         $FLAG[325] = $TIMER_FLAG[9] OR $FLAG[325]
      ;ENDFOLD
      ;FOLD -- RSK Fehlerausgabe K -- ;%{SE}%MKUKATPVW %CVW_COM %VCOMMENT %P 2:-- RSK Fehlerausgabe K --, 3: VW_COMMENT
      ;ENDFOLD
      ;FOLD F327 = !F832 & (A1105 & E1125 + !E1122) + F832 & (A1038 & E1108 + !E1025) + F327 ;%{SE}%MKUKATPVW %CVW_SPS %VBOASG %P 2:F327 = !F832 & (A1105 & E1125 + !E1122) + F832 & (A1038 & E1108 + !E1025) + F327, 3: BOASG
         $FLAG[327] = NOT $FLAG[832] AND ($OUT[1105] AND $IN[1125] OR NOT $IN[1122]) OR $FLAG[832] AND ($OUT[1038] AND $IN[1108] OR NOT $IN[1025]) OR $FLAG[327]
      ;ENDFOLD
      ;FOLD -- RSK Sammelstoerung -- ;%{SE}%MKUKATPVW %CVW_COM %VCOMMENT %P 2:-- RSK Sammelstoerung --, 3: VW_COMMENT
      ;ENDFOLD
      ;FOLD F329 = F325 + F326 + F327 ;%{SE}%MKUKATPVW %CVW_SPS %VBOASG %P 2:F329 = F325 + F326 + F327, 3: BOASG
         $FLAG[329] = $FLAG[325] OR $FLAG[326] OR $FLAG[327]
      ;ENDFOLD
      ;FOLD -- Kurzschlussschweissung SK3 -- ;%{SE}%MKUKATPVW %CVW_COM %VCOMMENT %P 2:-- Kurzschlussschweissung SK3 --, 3: VW_COMMENT
      ;ENDFOLD
      ;FOLD A1105 = (!F325 & !F329 & !F196 & !F830) + (F830 & A1105) ;%{SE}%MKUKATPVW %CVW_SPS %VBOASG %P 2:A1105 = (!F325 & !F329 & !F196 & !F830) + (F830 & A1105), 3: BOASG
         $OUT[1105] = (NOT $FLAG[325] AND NOT $FLAG[329] AND NOT $FLAG[196] AND NOT $FLAG[830]) OR ($FLAG[830] AND $OUT[1105])
      ;ENDFOLD
      ;FOLD F836 = AUS ;%{SE}%MKUKATPVW %CVW_SPS %VBOASG %P 2:F836 = AUS, 3: BOASG
         $FLAG[836] = FALSE
      ;ENDFOLD
      ;FOLD F836 = (E1039 & E1107 & !E1109 + E1039 & E15 + F326 + F327 + F122) & F830 & A4039 ;%{SE}%MKUKATPVW %CVW_SPS %VBOASG %P 2:F836 = (E1039 & E1107 & !E1109 + E1039 & E15 + F326 + F327 + F122) & F830 & A4039, 3: BOASG
         $FLAG[836] = ($IN[1039] AND $IN[1107] AND NOT $IN[1109] OR $IN[1039] AND $IN[15] OR $FLAG[326] OR $FLAG[327] OR $FLAG[122]) AND $FLAG[830] AND $OUT[4039]
      ;ENDFOLD
      ;FOLD -- Flagbildng Wiederholfraesen -- ;%{SE}%MKUKATPVW %CVW_COM %VCOMMENT %P 2:-- Flagbildng Wiederholfraesen --, 3: VW_COMMENT
      ;ENDFOLD
      ;FOLD F749 = (F322 + F323 + F325 + F326 + F327 + F329) & !F748 ;%{SE}%MKUKATPVW %CVW_SPS %VBOASG %P 2:F749 = (F322 + F323 + F325 + F326 + F327 + F329) & !F748, 3: BOASG
         $FLAG[749] = ($FLAG[322] OR $FLAG[323] OR $FLAG[325] OR $FLAG[326] OR $FLAG[327] OR $FLAG[329]) AND NOT $FLAG[748]
      ;ENDFOLD
      ;FOLD Schritt 118 = (E1105 & E1124 & !E1126 + E1105 & E15 + F326 + F327 + F196) & A4039 & !F832  ;%{SE}%MKUKATPVW %CVW_SPS %VST_CON %P 2:Schritt 118 = (E1105 & E1124 & !E1126 + E1105 & E15 + F326 + F327 + F196) & A4039 & !F832 , 3: ST_CON
         IF ($IN[1105] AND $IN[1124] AND NOT $IN[1126] OR $IN[1105] AND $IN[15] OR $FLAG[326] OR $FLAG[327] OR $FLAG[196]) AND $OUT[4039] AND NOT $FLAG[832] THEN
            PREVSTEP = $APP_INT[5]
            $APP_INT[5] = 118
         ENDIF
      ;ENDFOLD
      ;FOLD Schritt 118 = (E1039 & E1107 & !E1109 + E1039 & E15 + F326 + F327 + F196) & A4039 & F832  ;%{SE}%MKUKATPVW %CVW_SPS %VST_CON %P 2:Schritt 118 = (E1039 & E1107 & !E1109 + E1039 & E15 + F326 + F327 + F196) & A4039 & F832 , 3: ST_CON
         IF ($IN[1039] AND $IN[1107] AND NOT $IN[1109] OR $IN[1039] AND $IN[15] OR $FLAG[326] OR $FLAG[327] OR $FLAG[196]) AND $OUT[4039] AND $FLAG[832] THEN
            PREVSTEP = $APP_INT[5]
            $APP_INT[5] = 118
         ENDIF
      ;ENDFOLD
   ;ENDFOLD
   ;FOLD SCHRITT 118 -- STAT EZ3/SP3/KE3 -- ;%{P}%MKUKATPVW,%CSTEP,%VST_NR,%P 1:SCHRITT, 2:118, 3: STAT EZ3/SP3/KE3
      ;FOLD ;%{H}
         Case 118
      ;ENDFOLD
      ;FOLD F836 = AUS ;%{SE}%MKUKATPVW %CVW_SPS %VBOASG %P 2:F836 = AUS, 3: BOASG
         $FLAG[836] = FALSE
      ;ENDFOLD
      ;FOLD A1105 = F832 & A1105 ;%{SE}%MKUKATPVW %CVW_SPS %VBOASG %P 2:A1105 = F832 & A1105, 3: BOASG
         $OUT[1105] = $FLAG[832] AND $OUT[1105]
      ;ENDFOLD
      ;FOLD F174 = !F327 & F174 ;%{SE}%MKUKATPVW %CVW_SPS %VBOASG %P 2:F174 = !F327 & F174, 3: BOASG
         $FLAG[174] = NOT $FLAG[327] AND $FLAG[174]
      ;ENDFOLD
      ;FOLD F175 = F327 + F175 ;%{SE}%MKUKATPVW %CVW_SPS %VBOASG %P 2:F175 = F327 + F175, 3: BOASG
         $FLAG[175] = $FLAG[327] OR $FLAG[175]
      ;ENDFOLD
      ;FOLD -- EZ3/SP3/KE3 oeffnen -- ;%{SE}%MKUKATPVW %CVW_COM %VCOMMENT %P 2:-- EZ3/SP3/KE3 oeffnen --, 3: VW_COMMENT
      ;ENDFOLD
      ;FOLD A1039 = AUS ;%{SE}%MKUKATPVW %CVW_SPS %VBOASG %P 2:A1039 = AUS, 3: BOASG
         $OUT[1039] = FALSE
      ;ENDFOLD
      ;FOLD A1038 = AUS ;%{SE}%MKUKATPVW %CVW_SPS %VBOASG %P 2:A1038 = AUS, 3: BOASG
         $OUT[1038] = FALSE
      ;ENDFOLD
      ;FOLD A1037 = !E1037 ;%{SE}%MKUKATPVW %CVW_SPS %VBOASG %P 2:A1037 = !E1037, 3: BOASG
         $OUT[1037] = NOT $IN[1037]
      ;ENDFOLD
      ;FOLD -- Hilfsflag fuer KE3 -- ;%{SE}%MKUKATPVW %CVW_COM %VCOMMENT %P 2:-- Hilfsflag fuer KE3 --, 3: VW_COMMENT
      ;ENDFOLD
      ;FOLD F836 = !F326 & !F832 ;%{SE}%MKUKATPVW %CVW_SPS %VBOASG %P 2:F836 = !F326 & !F832, 3: BOASG
         $FLAG[836] = NOT $FLAG[326] AND NOT $FLAG[832]
      ;ENDFOLD
      ;FOLD bin9 ( F836 ) = 1 ;%{SE}%MKUKATPVW %CVW_SPS %VARIASG %P 2:bin9 ( F836 ) = 1, 3: ARIASG
         VW(#BINOUT,$FLAG[836],9,1)
      ;ENDFOLD
      ;FOLD -- Wartezeit Programmwechsel SK -- ;%{SE}%MKUKATPVW %CVW_COM %VCOMMENT %P 2:-- Wartezeit Programmwechsel SK --, 3: VW_COMMENT
      ;ENDFOLD
      ;FOLD T8 ( !F334 ) = -2[1/10Sek] ;%{SE}%MKUKATPVW %CVW_SPS %VTASG %P 2:T8 ( !F334 ) = -2[1/10Sek], 3: TASG
         VW(#SET_TIME,NOT $FLAG[334],8,0,-2)
      ;ENDFOLD
      ;FOLD -- Hilfsflag SK Programmwechsel -- ;%{SE}%MKUKATPVW %CVW_COM %VCOMMENT %P 2:-- Hilfsflag SK Programmwechsel --, 3: VW_COMMENT
      ;ENDFOLD
      ;FOLD F334 = EIN ;%{SE}%MKUKATPVW %CVW_SPS %VBOASG %P 2:F334 = EIN, 3: BOASG
         $FLAG[334] = TRUE
      ;ENDFOLD
      ;FOLD F748 = F322 + F323 + F325 + F326 + F327 + F329 ;%{SE}%MKUKATPVW %CVW_SPS %VBOASG %P 2:F748 = F322 + F323 + F325 + F326 + F327 + F329, 3: BOASG
         $FLAG[748] = $FLAG[322] OR $FLAG[323] OR $FLAG[325] OR $FLAG[326] OR $FLAG[327] OR $FLAG[329]
      ;ENDFOLD
      ;FOLD Schritt 97 = E1037 & !E1038 & (F322 + F323 + F325 + F326 + F327 + F329) & (E26 + E27) & A4039  ;%{SE}%MKUKATPVW %CVW_SPS %VST_CON %P 2:Schritt 97 = E1037 & !E1038 & (F322 + F323 + F325 + F326 + F327 + F329) & (E26 + E27) & A4039 , 3: ST_CON
         IF $IN[1037] AND NOT $IN[1038] AND ($FLAG[322] OR $FLAG[323] OR $FLAG[325] OR $FLAG[326] OR $FLAG[327] OR $FLAG[329]) AND ($IN[26] OR $IN[27]) AND $OUT[4039] THEN
            PREVSTEP = $APP_INT[5]
            $APP_INT[5] = 97
         ENDIF
      ;ENDFOLD
      ;FOLD Schritt 97 = E1037 & !E1038 & (F322 + F323 + F325 + F326 + F327 + F329) & (F731 & F749) & A4039  ;%{SE}%MKUKATPVW %CVW_SPS %VST_CON %P 2:Schritt 97 = E1037 & !E1038 & (F322 + F323 + F325 + F326 + F327 + F329) & (F731 & F749) & A4039 , 3: ST_CON
         IF $IN[1037] AND NOT $IN[1038] AND ($FLAG[322] OR $FLAG[323] OR $FLAG[325] OR $FLAG[326] OR $FLAG[327] OR $FLAG[329]) AND ($FLAG[731] AND $FLAG[749]) AND $OUT[4039] THEN
            PREVSTEP = $APP_INT[5]
            $APP_INT[5] = 97
         ENDIF
      ;ENDFOLD
      ;FOLD Schritt 119 = T8 & E1037 & !E1038 & (!F325 & !F329 & !F326 & !F327 + F196) & A4039  ;%{SE}%MKUKATPVW %CVW_SPS %VST_CON %P 2:Schritt 119 = T8 & E1037 & !E1038 & (!F325 & !F329 & !F326 & !F327 + F196) & A4039 , 3: ST_CON
         IF $TIMER_FLAG[8] AND $IN[1037] AND NOT $IN[1038] AND (NOT $FLAG[325] AND NOT $FLAG[329] AND NOT $FLAG[326] AND NOT $FLAG[327] OR $FLAG[196]) AND $OUT[4039] THEN
            PREVSTEP = $APP_INT[5]
            $APP_INT[5] = 119
         ENDIF
      ;ENDFOLD
   ;ENDFOLD
   ;FOLD SCHRITT 119 -- STAT EZ3/SP3/KE3 # Ende -- ;%{P}%MKUKATPVW,%CSTEP,%VST_NR,%P 1:SCHRITT, 2:119, 3: STAT EZ3/SP3/KE3 # Ende
      ;FOLD ;%{H}
         Case 119
      ;ENDFOLD
      ;FOLD -- Hilfsflag SK Programmwechsel -- ;%{SE}%MKUKATPVW %CVW_COM %VCOMMENT %P 2:-- Hilfsflag SK Programmwechsel --, 3: VW_COMMENT
      ;ENDFOLD
      ;FOLD F334 = AUS ;%{SE}%MKUKATPVW %CVW_SPS %VBOASG %P 2:F334 = AUS, 3: BOASG
         $FLAG[334] = FALSE
      ;ENDFOLD
      ;FOLD A116 = AUS ;%{SE}%MKUKATPVW %CVW_SPS %VBOASG %P 2:A116 = AUS, 3: BOASG
         $OUT[116] = FALSE
      ;ENDFOLD
      ;FOLD A194 = AUS ;%{SE}%MKUKATPVW %CVW_SPS %VBOASG %P 2:A194 = AUS, 3: BOASG
         $OUT[194] = FALSE
      ;ENDFOLD
      ;FOLD -- RSK Sammelstoerung -- ;%{SE}%MKUKATPVW %CVW_COM %VCOMMENT %P 2:-- RSK Sammelstoerung --, 3: VW_COMMENT
      ;ENDFOLD
      ;FOLD F329 = F196 ;%{SE}%MKUKATPVW %CVW_SPS %VBOASG %P 2:F329 = F196, 3: BOASG
         $FLAG[329] = $FLAG[196]
      ;ENDFOLD
      ;FOLD F185 = (!E1106 & !E1108 & !F832) + (!E1042 & !E1043 & F832) + F196 & (E26 + E27) ;%{SE}%MKUKATPVW %CVW_SPS %VBOASG %P 2:F185 = (!E1106 & !E1108 & !F832) + (!E1042 & !E1043 & F832) + F196 & (E26 + E27), 3: BOASG
         $FLAG[185] = (NOT $IN[1106] AND NOT $IN[1108] AND NOT $FLAG[832]) OR (NOT $IN[1042] AND NOT $IN[1043] AND $FLAG[832]) OR $FLAG[196] AND ($IN[26] OR $IN[27])
      ;ENDFOLD
      ;FOLD Schritt 1 = F185 & A4039  ;%{SE}%MKUKATPVW %CVW_SPS %VST_CON %P 2:Schritt 1 = F185 & A4039 , 3: ST_CON
         IF $FLAG[185] AND $OUT[4039] THEN
            PREVSTEP = $APP_INT[5]
            $APP_INT[5] = 1
         ENDIF
      ;ENDFOLD
   ;ENDFOLD
   ;FOLD SCHRITT 120 -- ROB STP1 SZ1 # Start -- ;%{P}%MKUKATPVW,%CSTEP,%VST_NR,%P 1:SCHRITT, 2:120, 3: ROB STP1 SZ1 # Start
      ;FOLD ;%{H}
         Case 120
      ;ENDFOLD
      ;FOLD -- RSK gestartet -- ;%{SE}%MKUKATPVW %CVW_COM %VCOMMENT %P 2:-- RSK gestartet --, 3: VW_COMMENT
      ;ENDFOLD
      ;FOLD F321 = AUS ;%{SE}%MKUKATPVW %CVW_SPS %VBOASG %P 2:F321 = AUS, 3: BOASG
         $FLAG[321] = FALSE
      ;ENDFOLD
      ;FOLD F122 = AUS ;%{SE}%MKUKATPVW %CVW_SPS %VBOASG %P 2:F122 = AUS, 3: BOASG
         $FLAG[122] = FALSE
      ;ENDFOLD
      ;FOLD F322 = AUS ;%{SE}%MKUKATPVW %CVW_SPS %VBOASG %P 2:F322 = AUS, 3: BOASG
         $FLAG[322] = FALSE
      ;ENDFOLD
      ;FOLD F323 = AUS ;%{SE}%MKUKATPVW %CVW_SPS %VBOASG %P 2:F323 = AUS, 3: BOASG
         $FLAG[323] = FALSE
      ;ENDFOLD
      ;FOLD F324 = AUS ;%{SE}%MKUKATPVW %CVW_SPS %VBOASG %P 2:F324 = AUS, 3: BOASG
         $FLAG[324] = FALSE
      ;ENDFOLD
      ;FOLD F325 = AUS ;%{SE}%MKUKATPVW %CVW_SPS %VBOASG %P 2:F325 = AUS, 3: BOASG
         $FLAG[325] = FALSE
      ;ENDFOLD
      ;FOLD F329 = AUS ;%{SE}%MKUKATPVW %CVW_SPS %VBOASG %P 2:F329 = AUS, 3: BOASG
         $FLAG[329] = FALSE
      ;ENDFOLD
      ;FOLD -- EZ1/SP1/STP1 SZ1 Zaehler -- ;%{SE}%MKUKATPVW %CVW_COM %VCOMMENT %P 2:-- EZ1/SP1/STP1 SZ1 Zaehler --, 3: VW_COMMENT
      ;ENDFOLD
      ;FOLD F94 = AUS ;%{SE}%MKUKATPVW %CVW_SPS %VBOASG %P 2:F94 = AUS, 3: BOASG
         $FLAG[94] = FALSE
      ;ENDFOLD
      ;FOLD F95 = AUS ;%{SE}%MKUKATPVW %CVW_SPS %VBOASG %P 2:F95 = AUS, 3: BOASG
         $FLAG[95] = FALSE
      ;ENDFOLD
      ;FOLD F96 = AUS ;%{SE}%MKUKATPVW %CVW_SPS %VBOASG %P 2:F96 = AUS, 3: BOASG
         $FLAG[96] = FALSE
      ;ENDFOLD
      ;FOLD F97 = AUS ;%{SE}%MKUKATPVW %CVW_SPS %VBOASG %P 2:F97 = AUS, 3: BOASG
         $FLAG[97] = FALSE
      ;ENDFOLD
      ;FOLD F98 = AUS ;%{SE}%MKUKATPVW %CVW_SPS %VBOASG %P 2:F98 = AUS, 3: BOASG
         $FLAG[98] = FALSE
      ;ENDFOLD
      ;FOLD F99 = AUS ;%{SE}%MKUKATPVW %CVW_SPS %VBOASG %P 2:F99 = AUS, 3: BOASG
         $FLAG[99] = FALSE
      ;ENDFOLD
      ;FOLD -- Hilfsflags Funktionstest KF Motor -- ;%{SE}%MKUKATPVW %CVW_COM %VCOMMENT %P 2:-- Hilfsflags Funktionstest KF Motor --, 3: VW_COMMENT
      ;ENDFOLD
      ;FOLD F312 = AUS ;%{SE}%MKUKATPVW %CVW_SPS %VBOASG %P 2:F312 = AUS, 3: BOASG
         $FLAG[312] = FALSE
      ;ENDFOLD
      ;FOLD F313 = AUS ;%{SE}%MKUKATPVW %CVW_SPS %VBOASG %P 2:F313 = AUS, 3: BOASG
         $FLAG[313] = FALSE
      ;ENDFOLD
      ;FOLD -- Rob. STP1 SZ1 beim Fraesen -- ;%{SE}%MKUKATPVW %CVW_COM %VCOMMENT %P 2:-- Rob. STP1 SZ1 beim Fraesen --, 3: VW_COMMENT
      ;ENDFOLD
      ;FOLD A116 = EIN ;%{SE}%MKUKATPVW %CVW_SPS %VBOASG %P 2:A116 = EIN, 3: BOASG
         $OUT[116] = TRUE
      ;ENDFOLD
      ;FOLD A130 = EIN ;%{SE}%MKUKATPVW %CVW_SPS %VBOASG %P 2:A130 = EIN, 3: BOASG
         $OUT[130] = TRUE
      ;ENDFOLD
      ;FOLD -- Ueberwachungszeit KF1 hochfahren -- ;%{SE}%MKUKATPVW %CVW_COM %VCOMMENT %P 2:-- Ueberwachungszeit KF1 hochfahren --, 3: VW_COMMENT
      ;ENDFOLD
      ;FOLD t8 ( EIN ) = -50[1/10Sek] ;%{SE}%MKUKATPVW %CVW_SPS %VTASG %P 2:t8 ( EIN ) = -50[1/10Sek], 3: TASG
         VW(#SET_TIME,TRUE,8,0,-50)
      ;ENDFOLD
      ;FOLD Schritt 121 = A4039  ;%{SE}%MKUKATPVW %CVW_SPS %VST_CON %P 2:Schritt 121 = A4039 , 3: ST_CON
         IF $OUT[4039] THEN
            PREVSTEP = $APP_INT[5]
            $APP_INT[5] = 121
         ENDIF
      ;ENDFOLD
   ;ENDFOLD
   ;FOLD SCHRITT 121 -- ROB STP1 SZ1 -- ;%{P}%MKUKATPVW,%CSTEP,%VST_NR,%P 1:SCHRITT, 2:121, 3: ROB STP1 SZ1
      ;FOLD ;%{H}
         Case 121
      ;ENDFOLD
      ;FOLD -- Umdreh. KF setzen -- ;%{SE}%MKUKATPVW %CVW_COM %VCOMMENT %P 2:-- Umdreh. KF setzen --, 3: VW_COMMENT
      ;ENDFOLD
      ;FOLD i1 ( EIN ) = 0 ;%{SE}%MKUKATPVW %CVW_SPS %VARIASG %P 2:i1 ( EIN ) = 0, 3: ARIASG
         VW(#COUNTER,TRUE,1,0)
      ;ENDFOLD
      ;FOLD -- Ueberwachungszeit KF1 -- ;%{SE}%MKUKATPVW %CVW_COM %VCOMMENT %P 2:-- Ueberwachungszeit KF1 --, 3: VW_COMMENT
      ;ENDFOLD
      ;FOLD t7 ( EIN ) = -60[1/10Sek] ;%{SE}%MKUKATPVW %CVW_SPS %VTASG %P 2:t7 ( EIN ) = -60[1/10Sek], 3: TASG
         VW(#SET_TIME,TRUE,7,0,-60)
      ;ENDFOLD
      ;FOLD -- KF1 einschalten -- ;%{SE}%MKUKATPVW %CVW_COM %VCOMMENT %P 2:-- KF1 einschalten --, 3: VW_COMMENT
      ;ENDFOLD
      ;FOLD i1 (EIN) = 0 ;%{SE}%MKUKATPVW %CVW_SPS %VARIASG %P 2:i1 (EIN) = 0, 3: ARIASG
         VW(#COUNTER,TRUE,1,0)
      ;ENDFOLD
      ;FOLD A864 = EIN ;%{SE}%MKUKATPVW %CVW_SPS %VBOASG %P 2:A864 = EIN, 3: BOASG
         $OUT[864] = TRUE
      ;ENDFOLD
      ;FOLD -- KF1 hochfahren -- ;%{SE}%MKUKATPVW %CVW_COM %VCOMMENT %P 2:-- KF1 hochfahren --, 3: VW_COMMENT
      ;ENDFOLD
      ;FOLD A863 = EIN ;%{SE}%MKUKATPVW %CVW_SPS %VBOASG %P 2:A863 = EIN, 3: BOASG
         $OUT[863] = TRUE
      ;ENDFOLD
      ;FOLD Schritt 122 = (!E863 + T8) & A4039  ;%{SE}%MKUKATPVW %CVW_SPS %VST_CON %P 2:Schritt 122 = (!E863 + T8) & A4039 , 3: ST_CON
         IF (NOT $IN[863] OR $TIMER_FLAG[8]) AND $OUT[4039] THEN
            PREVSTEP = $APP_INT[5]
            $APP_INT[5] = 122
         ENDIF
      ;ENDFOLD
   ;ENDFOLD
   ;FOLD SCHRITT 122 -- ROB STP1 SZ1 -- ;%{P}%MKUKATPVW,%CSTEP,%VST_NR,%P 1:SCHRITT, 2:122, 3: ROB STP1 SZ1
      ;FOLD ;%{H}
         Case 122
      ;ENDFOLD
      ;FOLD -- Funktionstest KF Motor -- ;%{SE}%MKUKATPVW %CVW_COM %VCOMMENT %P 2:-- Funktionstest KF Motor --, 3: VW_COMMENT
      ;ENDFOLD
      ;FOLD F312 = EIN ;%{SE}%MKUKATPVW %CVW_SPS %VBOASG %P 2:F312 = EIN, 3: BOASG
         $FLAG[312] = TRUE
      ;ENDFOLD
      ;FOLD F313 = i1 > 2 ;%{SE}%MKUKATPVW %CVW_SPS %VBOCMP %P 2:F313 = i1 > 2, 3: BOCMP
         $FLAG[313] = $COUNT_I[1] > 2
      ;ENDFOLD
      ;FOLD -- RSK Fehlerausgabe KF1 hochfahren -- ;%{SE}%MKUKATPVW %CVW_COM %VCOMMENT %P 2:-- RSK Fehlerausgabe KF1 hochfahren --, 3: VW_COMMENT
      ;ENDFOLD
      ;FOLD F324 = E863 + T8 + F324 ;%{SE}%MKUKATPVW %CVW_SPS %VBOASG %P 2:F324 = E863 + T8 + F324, 3: BOASG
         $FLAG[324] = $IN[863] OR $TIMER_FLAG[8] OR $FLAG[324]
      ;ENDFOLD
      ;FOLD Schritt 123 = (F313 + T7 + T8) & A4039  ;%{SE}%MKUKATPVW %CVW_SPS %VST_CON %P 2:Schritt 123 = (F313 + T7 + T8) & A4039 , 3: ST_CON
         IF ($FLAG[313] OR $TIMER_FLAG[7] OR $TIMER_FLAG[8]) AND $OUT[4039] THEN
            PREVSTEP = $APP_INT[5]
            $APP_INT[5] = 123
         ENDIF
      ;ENDFOLD
   ;ENDFOLD
   ;FOLD SCHRITT 123 -- ROB STP1 SZ1 -- ;%{P}%MKUKATPVW,%CSTEP,%VST_NR,%P 1:SCHRITT, 2:123, 3: ROB STP1 SZ1
      ;FOLD ;%{H}
         Case 123
      ;ENDFOLD
      ;FOLD F312 = AUS ;%{SE}%MKUKATPVW %CVW_SPS %VBOASG %P 2:F312 = AUS, 3: BOASG
         $FLAG[312] = FALSE
      ;ENDFOLD
      ;FOLD -- RSK Fehlerausgabe KF1 Initiator/Motor -- ;%{SE}%MKUKATPVW %CVW_COM %VCOMMENT %P 2:-- RSK Fehlerausgabe KF1 Initiator/Motor --, 3: VW_COMMENT
      ;ENDFOLD
      ;FOLD F322 = !F313 ;%{SE}%MKUKATPVW %CVW_SPS %VBOASG %P 2:F322 = !F313, 3: BOASG
         $FLAG[322] = NOT $FLAG[313]
      ;ENDFOLD
      ;FOLD -- Fraesfehler -- ;%{SE}%MKUKATPVW %CVW_COM %VCOMMENT %P 2:-- Fraesfehler --, 3: VW_COMMENT
      ;ENDFOLD
      ;FOLD F329 = F324 + F322 ;%{SE}%MKUKATPVW %CVW_SPS %VBOASG %P 2:F329 = F324 + F322, 3: BOASG
         $FLAG[329] = $FLAG[324] OR $FLAG[322]
      ;ENDFOLD
      ;FOLD -- Fraeser aus bei Fehler -- ;%{SE}%MKUKATPVW %CVW_COM %VCOMMENT %P 2:-- Fraeser aus bei Fehler --, 3: VW_COMMENT
      ;ENDFOLD
      ;FOLD A864 = !F329 ;%{SE}%MKUKATPVW %CVW_SPS %VBOASG %P 2:A864 = !F329, 3: BOASG
         $OUT[864] = NOT $FLAG[329]
      ;ENDFOLD
      ;FOLD -- Warte Fraesen fertig oder Timeout -- ;%{SE}%MKUKATPVW %CVW_COM %VCOMMENT %P 2:-- Warte Fraesen fertig oder Timeout --, 3: VW_COMMENT
      ;ENDFOLD
      ;FOLD Schritt 124 = (F79 & F98 + F78 & F94 & !F287 + T7) & A4039  ;%{SE}%MKUKATPVW %CVW_SPS %VST_CON %P 2:Schritt 124 = (F79 & F98 + F78 & F94 & !F287 + T7) & A4039 , 3: ST_CON
         IF ($FLAG[79] AND $FLAG[98] OR $FLAG[78] AND $FLAG[94] AND NOT $FLAG[287] OR $TIMER_FLAG[7]) AND $OUT[4039] THEN
            PREVSTEP = $APP_INT[5]
            $APP_INT[5] = 124
         ENDIF
      ;ENDFOLD
      ;FOLD Schritt 124 = (F78 & F96 & F287 + T7) & A4039  ;%{SE}%MKUKATPVW %CVW_SPS %VST_CON %P 2:Schritt 124 = (F78 & F96 & F287 + T7) & A4039 , 3: ST_CON
         IF ($FLAG[78] AND $FLAG[96] AND $FLAG[287] OR $TIMER_FLAG[7]) AND $OUT[4039] THEN
            PREVSTEP = $APP_INT[5]
            $APP_INT[5] = 124
         ENDIF
      ;ENDFOLD
   ;ENDFOLD
   ;FOLD SCHRITT 124 -- ROB STP1 SZ1 -- ;%{P}%MKUKATPVW,%CSTEP,%VST_NR,%P 1:SCHRITT, 2:124, 3: ROB STP1 SZ1
      ;FOLD ;%{H}
         Case 124
      ;ENDFOLD
      ;FOLD -- Hilfsflag SK Programmwechsel -- ;%{SE}%MKUKATPVW %CVW_COM %VCOMMENT %P 2:-- Hilfsflag SK Programmwechsel --, 3: VW_COMMENT
      ;ENDFOLD
      ;FOLD F334 = AUS ;%{SE}%MKUKATPVW %CVW_SPS %VBOASG %P 2:F334 = AUS, 3: BOASG
         $FLAG[334] = FALSE
      ;ENDFOLD
      ;FOLD -- KF1 runterfahren -- ;%{SE}%MKUKATPVW %CVW_COM %VCOMMENT %P 2:-- KF1 runterfahren --, 3: VW_COMMENT
      ;ENDFOLD
      ;FOLD A863 = AUS ;%{SE}%MKUKATPVW %CVW_SPS %VBOASG %P 2:A863 = AUS, 3: BOASG
         $OUT[863] = FALSE
      ;ENDFOLD
      ;FOLD -- Fraesfehler -- ;%{SE}%MKUKATPVW %CVW_COM %VCOMMENT %P 2:-- Fraesfehler --, 3: VW_COMMENT
      ;ENDFOLD
      ;FOLD F329 = T7 + F324 ;%{SE}%MKUKATPVW %CVW_SPS %VBOASG %P 2:F329 = T7 + F324, 3: BOASG
         $FLAG[329] = $TIMER_FLAG[7] OR $FLAG[324]
      ;ENDFOLD
      ;FOLD -- Hilfsflag Startfraesen -- ;%{SE}%MKUKATPVW %CVW_COM %VCOMMENT %P 2:-- Hilfsflag Startfraesen --, 3: VW_COMMENT
      ;ENDFOLD
      ;FOLD F96 = F96 & F287 ;%{SE}%MKUKATPVW %CVW_SPS %VBOASG %P 2:F96 = F96 & F287, 3: BOASG
         $FLAG[96] = $FLAG[96] AND $FLAG[287]
      ;ENDFOLD
      ;FOLD F287 = F78 ;%{SE}%MKUKATPVW %CVW_SPS %VBOASG %P 2:F287 = F78, 3: BOASG
         $FLAG[287] = $FLAG[78]
      ;ENDFOLD
      ;FOLD -- Wiederholung beim Startfraesen -- ;%{SE}%MKUKATPVW %CVW_COM %VCOMMENT %P 2:-- Wiederholung beim Startfraesen --, 3: VW_COMMENT
      ;ENDFOLD
      ;FOLD Schritt 121 = E863 & F78 & !F96 & !F329 & A4039  ;%{SE}%MKUKATPVW %CVW_SPS %VST_CON %P 2:Schritt 121 = E863 & F78 & !F96 & !F329 & A4039 , 3: ST_CON
         IF $IN[863] AND $FLAG[78] AND NOT $FLAG[96] AND NOT $FLAG[329] AND $OUT[4039] THEN
            PREVSTEP = $APP_INT[5]
            $APP_INT[5] = 121
         ENDIF
      ;ENDFOLD
      ;FOLD -- Weiter wenn Fraesen fertig -- ;%{SE}%MKUKATPVW %CVW_COM %VCOMMENT %P 2:-- Weiter wenn Fraesen fertig --, 3: VW_COMMENT
      ;ENDFOLD
      ;FOLD Schritt 125 = E863 & (F79 & F98 + F78 & F96 + F329) & A4039  ;%{SE}%MKUKATPVW %CVW_SPS %VST_CON %P 2:Schritt 125 = E863 & (F79 & F98 + F78 & F96 + F329) & A4039 , 3: ST_CON
         IF $IN[863] AND ($FLAG[79] AND $FLAG[98] OR $FLAG[78] AND $FLAG[96] OR $FLAG[329]) AND $OUT[4039] THEN
            PREVSTEP = $APP_INT[5]
            $APP_INT[5] = 125
         ENDIF
      ;ENDFOLD
      ;FOLD -- Weiter bei Fehler -- ;%{SE}%MKUKATPVW %CVW_COM %VCOMMENT %P 2:-- Weiter bei Fehler --, 3: VW_COMMENT
      ;ENDFOLD
      ;FOLD Schritt 127 = F329 & (E26 + E27) & A4039  ;%{SE}%MKUKATPVW %CVW_SPS %VST_CON %P 2:Schritt 127 = F329 & (E26 + E27) & A4039 , 3: ST_CON
         IF $FLAG[329] AND ($IN[26] OR $IN[27]) AND $OUT[4039] THEN
            PREVSTEP = $APP_INT[5]
            $APP_INT[5] = 127
         ENDIF
      ;ENDFOLD
   ;ENDFOLD
   ;FOLD SCHRITT 125 -- ROB STP1 SZ1 -- ;%{P}%MKUKATPVW,%CSTEP,%VST_NR,%P 1:SCHRITT, 2:125, 3: ROB STP1 SZ1
      ;FOLD ;%{H}
         Case 125
      ;ENDFOLD
      ;FOLD -- KF1 einschalten -- ;%{SE}%MKUKATPVW %CVW_COM %VCOMMENT %P 2:-- KF1 einschalten --, 3: VW_COMMENT
      ;ENDFOLD
      ;FOLD A864 = AUS ;%{SE}%MKUKATPVW %CVW_SPS %VBOASG %P 2:A864 = AUS, 3: BOASG
         $OUT[864] = FALSE
      ;ENDFOLD
      ;FOLD bin3 (!F329) = 1 ;%{SE}%MKUKATPVW %CVW_SPS %VARIASG %P 2:bin3 (!F329) = 1, 3: ARIASG
         VW(#BINOUT,NOT $FLAG[329],3,1)
      ;ENDFOLD
      ;FOLD -- Wartezeit Programmwechsel SK -- ;%{SE}%MKUKATPVW %CVW_COM %VCOMMENT %P 2:-- Wartezeit Programmwechsel SK --, 3: VW_COMMENT
      ;ENDFOLD
      ;FOLD T8 ( !F334 ) = -2[1/10Sek] ;%{SE}%MKUKATPVW %CVW_SPS %VTASG %P 2:T8 ( !F334 ) = -2[1/10Sek], 3: TASG
         VW(#SET_TIME,NOT $FLAG[334],8,0,-2)
      ;ENDFOLD
      ;FOLD -- Hilfsflag SK Programmwechsel -- ;%{SE}%MKUKATPVW %CVW_COM %VCOMMENT %P 2:-- Hilfsflag SK Programmwechsel --, 3: VW_COMMENT
      ;ENDFOLD
      ;FOLD F334 = EIN ;%{SE}%MKUKATPVW %CVW_SPS %VBOASG %P 2:F334 = EIN, 3: BOASG
         $FLAG[334] = TRUE
      ;ENDFOLD
      ;FOLD Schritt 126 = T8 & A4039  ;%{SE}%MKUKATPVW %CVW_SPS %VST_CON %P 2:Schritt 126 = T8 & A4039 , 3: ST_CON
         IF $TIMER_FLAG[8] AND $OUT[4039] THEN
            PREVSTEP = $APP_INT[5]
            $APP_INT[5] = 126
         ENDIF
      ;ENDFOLD
   ;ENDFOLD
   ;FOLD SCHRITT 126 -- ROB STP1 SZ1 -- ;%{P}%MKUKATPVW,%CSTEP,%VST_NR,%P 1:SCHRITT, 2:126, 3: ROB STP1 SZ1
      ;FOLD ;%{H}
         Case 126
      ;ENDFOLD
      ;FOLD -- Hilfsflag SK Programmwechsel -- ;%{SE}%MKUKATPVW %CVW_COM %VCOMMENT %P 2:-- Hilfsflag SK Programmwechsel --, 3: VW_COMMENT
      ;ENDFOLD
      ;FOLD F334 = AUS ;%{SE}%MKUKATPVW %CVW_SPS %VBOASG %P 2:F334 = AUS, 3: BOASG
         $FLAG[334] = FALSE
      ;ENDFOLD
      ;FOLD -- RSK Sammelstoerung -- ;%{SE}%MKUKATPVW %CVW_COM %VCOMMENT %P 2:-- RSK Sammelstoerung --, 3: VW_COMMENT
      ;ENDFOLD
      ;FOLD F329 = T7 ;%{SE}%MKUKATPVW %CVW_SPS %VBOASG %P 2:F329 = T7, 3: BOASG
         $FLAG[329] = $TIMER_FLAG[7]
      ;ENDFOLD
      ;FOLD -- Quitt. Fraesen SK1 -- ;%{SE}%MKUKATPVW %CVW_COM %VCOMMENT %P 2:-- Quitt. Fraesen SK1 --, 3: VW_COMMENT
      ;ENDFOLD
      ;FOLD A786 = !F329 & !F322 ;%{SE}%MKUKATPVW %CVW_SPS %VBOASG %P 2:A786 = !F329 & !F322, 3: BOASG
         $OUT[786] = NOT $FLAG[329] AND NOT $FLAG[322]
      ;ENDFOLD
      ;FOLD Schritt 127 = !E786 & E787 & !E788 & !F329  ;%{SE}%MKUKATPVW %CVW_SPS %VST_CON %P 2:Schritt 127 = !E786 & E787 & !E788 & !F329 , 3: ST_CON
         IF NOT $IN[786] AND $IN[787] AND NOT $IN[788] AND NOT $FLAG[329] THEN
            PREVSTEP = $APP_INT[5]
            $APP_INT[5] = 127
         ENDIF
      ;ENDFOLD
   ;ENDFOLD
   ;FOLD SCHRITT 127 -- ROB STP1 SZ1 # Ende -- ;%{P}%MKUKATPVW,%CSTEP,%VST_NR,%P 1:SCHRITT, 2:127, 3: ROB STP1 SZ1 # Ende
      ;FOLD ;%{H}
         Case 127
      ;ENDFOLD
      ;FOLD -- RSK Sammelstoerung -- ;%{SE}%MKUKATPVW %CVW_COM %VCOMMENT %P 2:-- RSK Sammelstoerung --, 3: VW_COMMENT
      ;ENDFOLD
      ;FOLD F329 = T7 ;%{SE}%MKUKATPVW %CVW_SPS %VBOASG %P 2:F329 = T7, 3: BOASG
         $FLAG[329] = $TIMER_FLAG[7]
      ;ENDFOLD
      ;FOLD F91 = !F329 ;%{SE}%MKUKATPVW %CVW_SPS %VBOASG %P 2:F91 = !F329, 3: BOASG
         $FLAG[91] = NOT $FLAG[329]
      ;ENDFOLD
      ;FOLD Schritt 120 = F329 & (E26 + E27) & A4039  ;%{SE}%MKUKATPVW %CVW_SPS %VST_CON %P 2:Schritt 120 = F329 & (E26 + E27) & A4039 , 3: ST_CON
         IF $FLAG[329] AND ($IN[26] OR $IN[27]) AND $OUT[4039] THEN
            PREVSTEP = $APP_INT[5]
            $APP_INT[5] = 120
         ENDIF
      ;ENDFOLD
      ;FOLD Schritt 1 = F91 & !F329 & A4039  ;%{SE}%MKUKATPVW %CVW_SPS %VST_CON %P 2:Schritt 1 = F91 & !F329 & A4039 , 3: ST_CON
         IF $FLAG[91] AND NOT $FLAG[329] AND $OUT[4039] THEN
            PREVSTEP = $APP_INT[5]
            $APP_INT[5] = 1
         ENDIF
      ;ENDFOLD
   ;ENDFOLD
   ;FOLD SCHRITT 128 -- MS1 Reinigung (an KS3)-- ;%{P}%MKUKATPVW,%CSTEP,%VST_NR,%P 1:SCHRITT, 2:128, 3: MS1 Reinigung (an KS3)
      ;FOLD ;%{H}
         Case 128
      ;ENDFOLD
      ;FOLD -- RSK gestartet -- ;%{SE}%MKUKATPVW %CVW_COM %VCOMMENT %P 2:-- RSK gestartet --, 3: VW_COMMENT
      ;ENDFOLD
      ;FOLD F321 = AUS ;%{SE}%MKUKATPVW %CVW_SPS %VBOASG %P 2:F321 = AUS, 3: BOASG
         $FLAG[321] = FALSE
      ;ENDFOLD
      ;FOLD F323 = AUS ;%{SE}%MKUKATPVW %CVW_SPS %VBOASG %P 2:F323 = AUS, 3: BOASG
         $FLAG[323] = FALSE
      ;ENDFOLD
      ;FOLD F324 = AUS ;%{SE}%MKUKATPVW %CVW_SPS %VBOASG %P 2:F324 = AUS, 3: BOASG
         $FLAG[324] = FALSE
      ;ENDFOLD
      ;FOLD F329 = AUS ;%{SE}%MKUKATPVW %CVW_SPS %VBOASG %P 2:F329 = AUS, 3: BOASG
         $FLAG[329] = FALSE
      ;ENDFOLD
      ;FOLD -- MS1 Reinigung gestartet -- ;%{SE}%MKUKATPVW %CVW_COM %VCOMMENT %P 2:-- MS1 Reinigung gestartet --, 3: VW_COMMENT
      ;ENDFOLD
      ;FOLD F604 = EIN ;%{SE}%MKUKATPVW %CVW_SPS %VBOASG %P 2:F604 = EIN, 3: BOASG
         $FLAG[604] = TRUE
      ;ENDFOLD
      ;FOLD -- MS bei Reinigung -- ;%{SE}%MKUKATPVW %CVW_COM %VCOMMENT %P 2:-- MS bei Reinigung --, 3: VW_COMMENT
      ;ENDFOLD
      ;FOLD A116 = EIN ;%{SE}%MKUKATPVW %CVW_SPS %VBOASG %P 2:A116 = EIN, 3: BOASG
         $OUT[116] = TRUE
      ;ENDFOLD
      ;FOLD -- Ueberwachungszeit KS3 schwenken -- ;%{SE}%MKUKATPVW %CVW_COM %VCOMMENT %P 2:-- Ueberwachungszeit KS3 schwenken --, 3: VW_COMMENT
      ;ENDFOLD
      ;FOLD t8 ( EIN ) = -100[1/10Sek] ;%{SE}%MKUKATPVW %CVW_SPS %VTASG %P 2:t8 ( EIN ) = -100[1/10Sek], 3: TASG
         VW(#SET_TIME,TRUE,8,0,-100)
      ;ENDFOLD
      ;FOLD Schritt 129 = A4039  ;%{SE}%MKUKATPVW %CVW_SPS %VST_CON %P 2:Schritt 129 = A4039 , 3: ST_CON
         IF $OUT[4039] THEN
            PREVSTEP = $APP_INT[5]
            $APP_INT[5] = 129
         ENDIF
      ;ENDFOLD
   ;ENDFOLD
   ;FOLD SCHRITT 129 -- MS1 Reinigung (an KS3) -- ;%{P}%MKUKATPVW,%CSTEP,%VST_NR,%P 1:SCHRITT, 2:129, 3: MS1 Reinigung (an KS3)
      ;FOLD ;%{H}
         Case 129
      ;ENDFOLD
      ;FOLD -- RSK Fehlerausgabe KS3 Ruhest. -- ;%{SE}%MKUKATPVW %CVW_COM %VCOMMENT %P 2:-- RSK Fehlerausgabe KS3 Ruhest. --, 3: VW_COMMENT
      ;ENDFOLD
      ;FOLD F323 = !E1162 ;%{SE}%MKUKATPVW %CVW_SPS %VBOASG %P 2:F323 = !E1162, 3: BOASG
         $FLAG[323] = NOT $IN[1162]
      ;ENDFOLD
      ;FOLD -- RSK Sammelstoerung -- ;%{SE}%MKUKATPVW %CVW_COM %VCOMMENT %P 2:-- RSK Sammelstoerung --, 3: VW_COMMENT
      ;ENDFOLD
      ;FOLD F329 = F323 ;%{SE}%MKUKATPVW %CVW_SPS %VBOASG %P 2:F329 = F323, 3: BOASG
         $FLAG[329] = $FLAG[323]
      ;ENDFOLD
      ;FOLD Schritt 128 = (E26 + E27) & F323 & A4039  ;%{SE}%MKUKATPVW %CVW_SPS %VST_CON %P 2:Schritt 128 = (E26 + E27) & F323 & A4039 , 3: ST_CON
         IF ($IN[26] OR $IN[27]) AND $FLAG[323] AND $OUT[4039] THEN
            PREVSTEP = $APP_INT[5]
            $APP_INT[5] = 128
         ENDIF
      ;ENDFOLD
      ;FOLD Schritt 130 = (!F323 + T8) & A4039  ;%{SE}%MKUKATPVW %CVW_SPS %VST_CON %P 2:Schritt 130 = (!F323 + T8) & A4039 , 3: ST_CON
         IF (NOT $FLAG[323] OR $TIMER_FLAG[8]) AND $OUT[4039] THEN
            PREVSTEP = $APP_INT[5]
            $APP_INT[5] = 130
         ENDIF
      ;ENDFOLD
   ;ENDFOLD
   ;FOLD SCHRITT 130 -- MS1 Reinigung (an KS3) -- ;%{P}%MKUKATPVW,%CSTEP,%VST_NR,%P 1:SCHRITT, 2:130, 3: MS1 Reinigung (an KS3)
      ;FOLD ;%{H}
         Case 130
      ;ENDFOLD
      ;FOLD -- KS3 in Arbeitsstellung schwenken -- ;%{SE}%MKUKATPVW %CVW_COM %VCOMMENT %P 2:-- KS3 in Arbeitsstellung schwenken --, 3: VW_COMMENT
      ;ENDFOLD
      ;FOLD A1162 = !E1163 ;%{SE}%MKUKATPVW %CVW_SPS %VBOASG %P 2:A1162 = !E1163, 3: BOASG
         $OUT[1162] = NOT $IN[1163]
      ;ENDFOLD
      ;FOLD Schritt 131 = A4039  ;%{SE}%MKUKATPVW %CVW_SPS %VST_CON %P 2:Schritt 131 = A4039 , 3: ST_CON
         IF $OUT[4039] THEN
            PREVSTEP = $APP_INT[5]
            $APP_INT[5] = 131
         ENDIF
      ;ENDFOLD
   ;ENDFOLD
   ;FOLD SCHRITT 131 -- MS1 Reinigung (an KS3) -- ;%{P}%MKUKATPVW,%CSTEP,%VST_NR,%P 1:SCHRITT, 2:131, 3: MS1 Reinigung (an KS3)
      ;FOLD ;%{H}
         Case 131
      ;ENDFOLD
      ;FOLD -- RSK Fehlerausgabe KS3 Arbeitsstellung -- ;%{SE}%MKUKATPVW %CVW_COM %VCOMMENT %P 2:-- RSK Fehlerausgabe KS3 Arbeitsstellung --, 3: VW_COMMENT
      ;ENDFOLD
      ;FOLD F324 = !E1163 & T8 + F324 ;%{SE}%MKUKATPVW %CVW_SPS %VBOASG %P 2:F324 = !E1163 & T8 + F324, 3: BOASG
         $FLAG[324] = NOT $IN[1163] AND $TIMER_FLAG[8] OR $FLAG[324]
      ;ENDFOLD
      ;FOLD -- RSK Sammelstoerung -- ;%{SE}%MKUKATPVW %CVW_COM %VCOMMENT %P 2:-- RSK Sammelstoerung --, 3: VW_COMMENT
      ;ENDFOLD
      ;FOLD F329 = F324 ;%{SE}%MKUKATPVW %CVW_SPS %VBOASG %P 2:F329 = F324, 3: BOASG
         $FLAG[329] = $FLAG[324]
      ;ENDFOLD
      ;FOLD Schritt 128 = F324 & (E26 + E27) & A4039  ;%{SE}%MKUKATPVW %CVW_SPS %VST_CON %P 2:Schritt 128 = F324 & (E26 + E27) & A4039 , 3: ST_CON
         IF $FLAG[324] AND ($IN[26] OR $IN[27]) AND $OUT[4039] THEN
            PREVSTEP = $APP_INT[5]
            $APP_INT[5] = 128
         ENDIF
      ;ENDFOLD
      ;FOLD Schritt 132 = !F324 & E1163 & !E1165 & A4039  ;%{SE}%MKUKATPVW %CVW_SPS %VST_CON %P 2:Schritt 132 = !F324 & E1163 & !E1165 & A4039 , 3: ST_CON
         IF NOT $FLAG[324] AND $IN[1163] AND NOT $IN[1165] AND $OUT[4039] THEN
            PREVSTEP = $APP_INT[5]
            $APP_INT[5] = 132
         ENDIF
      ;ENDFOLD
   ;ENDFOLD
   ;FOLD SCHRITT 132 -- MS1 Reinigung (an KS3) -- ;%{P}%MKUKATPVW,%CSTEP,%VST_NR,%P 1:SCHRITT, 2:132, 3: MS1 Reinigung (an KS3)
      ;FOLD ;%{H}
         Case 132
      ;ENDFOLD
      ;FOLD A1864 = AUS ;%{SE}%MKUKATPVW %CVW_SPS %VBOASG %P 2:A1864 = AUS, 3: BOASG
         $OUT[1864] = FALSE
      ;ENDFOLD
      ;FOLD A2168 = AUS ;%{SE}%MKUKATPVW %CVW_SPS %VBOASG %P 2:A2168 = AUS, 3: BOASG
         $OUT[2168] = FALSE
      ;ENDFOLD
      ;FOLD -- Ueberwachungszeit Versetzeinheit -- ;%{SE}%MKUKATPVW %CVW_COM %VCOMMENT %P 2:-- Ueberwachungszeit Versetzeinheit --, 3: VW_COMMENT
      ;ENDFOLD
      ;FOLD t8 ( EIN ) = -50[1/10Sek] ;%{SE}%MKUKATPVW %CVW_SPS %VTASG %P 2:t8 ( EIN ) = -50[1/10Sek], 3: TASG
         VW(#SET_TIME,TRUE,8,0,-50)
      ;ENDFOLD
      ;FOLD -- Ueberwachungszeit Reinigung -- ;%{SE}%MKUKATPVW %CVW_COM %VCOMMENT %P 2:-- Ueberwachungszeit Reinigung --, 3: VW_COMMENT
      ;ENDFOLD
      ;FOLD t9 ( EIN ) = -80[1/10Sek] ;%{SE}%MKUKATPVW %CVW_SPS %VTASG %P 2:t9 ( EIN ) = -80[1/10Sek], 3: TASG
         VW(#SET_TIME,TRUE,9,0,-80)
      ;ENDFOLD
      ;FOLD Schritt 133 = A4039  ;%{SE}%MKUKATPVW %CVW_SPS %VST_CON %P 2:Schritt 133 = A4039 , 3: ST_CON
         IF $OUT[4039] THEN
            PREVSTEP = $APP_INT[5]
            $APP_INT[5] = 133
         ENDIF
      ;ENDFOLD
   ;ENDFOLD
   ;FOLD SCHRITT 133 -- MS1 Reinigung (an KS3) -- ;%{P}%MKUKATPVW,%CSTEP,%VST_NR,%P 1:SCHRITT, 2:133, 3: MS1 Reinigung (an KS3)
      ;FOLD ;%{H}
         Case 133
      ;ENDFOLD
      ;FOLD -- RSK Fehlerausgabe Versetzeinheit -- ;%{SE}%MKUKATPVW %CVW_COM %VCOMMENT %P 2:-- RSK Fehlerausgabe Versetzeinheit --, 3: VW_COMMENT
      ;ENDFOLD
      ;FOLD F328 = F576 & T8 ;%{SE}%MKUKATPVW %CVW_SPS %VBOASG %P 2:F328 = F576 & T8, 3: BOASG
         $FLAG[328] = $FLAG[576] AND $TIMER_FLAG[8]
      ;ENDFOLD
      ;FOLD -- RSK Sammelstoerung -- ;%{SE}%MKUKATPVW %CVW_COM %VCOMMENT %P 2:-- RSK Sammelstoerung --, 3: VW_COMMENT
      ;ENDFOLD
      ;FOLD F329 = T8 ;%{SE}%MKUKATPVW %CVW_SPS %VBOASG %P 2:F329 = T8, 3: BOASG
         $FLAG[329] = $TIMER_FLAG[8]
      ;ENDFOLD
      ;FOLD -- Zeit Reinigung LZ -- ;%{SE}%MKUKATPVW %CVW_COM %VCOMMENT %P 2:-- Zeit Reinigung LZ --, 3: VW_COMMENT
      ;ENDFOLD
      ;FOLD F271 = i26 = 0 ;%{SE}%MKUKATPVW %CVW_SPS %VBOCMP %P 2:F271 = i26 = 0, 3: BOCMP
         $FLAG[271] = $COUNT_I[26] == 0
      ;ENDFOLD
      ;FOLD t7 ( F271 ) = -20[1/10Sek] ;%{SE}%MKUKATPVW %CVW_SPS %VTASG %P 2:t7 ( F271 ) = -20[1/10Sek], 3: TASG
         VW(#SET_TIME,$FLAG[271],7,0,-20)
      ;ENDFOLD
      ;FOLD t7 ( !F271 ) = i26[1/10Sek] ;%{SE}%MKUKATPVW %CVW_SPS %VTASG %P 2:t7 ( !F271 ) = i26[1/10Sek], 3: TASG
         VW(#SET_TIME,NOT $FLAG[271],7,0,$COUNT_I[26])
      ;ENDFOLD
      ;FOLD -- Versetzeinheit in Arbeitsst. schw. -- ;%{SE}%MKUKATPVW %CVW_COM %VCOMMENT %P 2:-- Versetzeinheit in Arbeitsst. schw. --, 3: VW_COMMENT
      ;ENDFOLD
      ;FOLD A2168 = !E2168 & F576 ;%{SE}%MKUKATPVW %CVW_SPS %VBOASG %P 2:A2168 = !E2168 & F576, 3: BOASG
         $OUT[2168] = NOT $IN[2168] AND $FLAG[576]
      ;ENDFOLD
      ;FOLD Schritt 132 = A2168 & T8 & (E26 + E27) & A4039  ;%{SE}%MKUKATPVW %CVW_SPS %VST_CON %P 2:Schritt 132 = A2168 & T8 & (E26 + E27) & A4039 , 3: ST_CON
         IF $OUT[2168] AND $TIMER_FLAG[8] AND ($IN[26] OR $IN[27]) AND $OUT[4039] THEN
            PREVSTEP = $APP_INT[5]
            $APP_INT[5] = 132
         ENDIF
      ;ENDFOLD
      ;FOLD Schritt 134 = (E2168 & F576 + !E2168 & !F576) & A4039  ;%{SE}%MKUKATPVW %CVW_SPS %VST_CON %P 2:Schritt 134 = (E2168 & F576 + !E2168 & !F576) & A4039 , 3: ST_CON
         IF ($IN[2168] AND $FLAG[576] OR NOT $IN[2168] AND NOT $FLAG[576]) AND $OUT[4039] THEN
            PREVSTEP = $APP_INT[5]
            $APP_INT[5] = 134
         ENDIF
      ;ENDFOLD
   ;ENDFOLD
   ;FOLD SCHRITT 134 -- MS1 Reinigung (an KS3) -- ;%{P}%MKUKATPVW,%CSTEP,%VST_NR,%P 1:SCHRITT, 2:134, 3: MS1 Reinigung (an KS3)
      ;FOLD ;%{H}
         Case 134
      ;ENDFOLD
      ;FOLD -- RSK Sammelstoerung -- ;%{SE}%MKUKATPVW %CVW_COM %VCOMMENT %P 2:-- RSK Sammelstoerung --, 3: VW_COMMENT
      ;ENDFOLD
      ;FOLD F329 = T9 ;%{SE}%MKUKATPVW %CVW_SPS %VBOASG %P 2:F329 = T9, 3: BOASG
         $FLAG[329] = $TIMER_FLAG[9]
      ;ENDFOLD
      ;FOLD -- MS1 Ausblasen EIN -- ;%{SE}%MKUKATPVW %CVW_COM %VCOMMENT %P 2:-- MS1 Ausblasen EIN --, 3: VW_COMMENT
      ;ENDFOLD
      ;FOLD A1870 = EIN ;%{SE}%MKUKATPVW %CVW_SPS %VBOASG %P 2:A1870 = EIN, 3: BOASG
         $OUT[1870] = TRUE
      ;ENDFOLD
      ;FOLD -- MS1 Reinigung starten -- ;%{SE}%MKUKATPVW %CVW_COM %VCOMMENT %P 2:-- MS1 Reinigung starten --, 3: VW_COMMENT
      ;ENDFOLD
      ;FOLD A1864 = EIN ;%{SE}%MKUKATPVW %CVW_SPS %VBOASG %P 2:A1864 = EIN, 3: BOASG
         $OUT[1864] = TRUE
      ;ENDFOLD
      ;FOLD Schritt 132 = (!E1864 + E1864 & !F271) & T9 & (E26 + E27) & A4039  ;%{SE}%MKUKATPVW %CVW_SPS %VST_CON %P 2:Schritt 132 = (!E1864 + E1864 & !F271) & T9 & (E26 + E27) & A4039 , 3: ST_CON
         IF (NOT $IN[1864] OR $IN[1864] AND NOT $FLAG[271]) AND $TIMER_FLAG[9] AND ($IN[26] OR $IN[27]) AND $OUT[4039] THEN
            PREVSTEP = $APP_INT[5]
            $APP_INT[5] = 132
         ENDIF
      ;ENDFOLD
      ;FOLD Schritt 135 = (E1864 + !E1864 & !F271 & T7) & A4039  ;%{SE}%MKUKATPVW %CVW_SPS %VST_CON %P 2:Schritt 135 = (E1864 + !E1864 & !F271 & T7) & A4039 , 3: ST_CON
         IF ($IN[1864] OR NOT $IN[1864] AND NOT $FLAG[271] AND $TIMER_FLAG[7]) AND $OUT[4039] THEN
            PREVSTEP = $APP_INT[5]
            $APP_INT[5] = 135
         ENDIF
      ;ENDFOLD
   ;ENDFOLD
   ;FOLD SCHRITT 135 -- MS1 Reinigung (an KS3) -- ;%{P}%MKUKATPVW,%CSTEP,%VST_NR,%P 1:SCHRITT, 2:135, 3: MS1 Reinigung (an KS3)
      ;FOLD ;%{H}
         Case 135
      ;ENDFOLD
      ;FOLD -- MS1 Reinigung beenden -- ;%{SE}%MKUKATPVW %CVW_COM %VCOMMENT %P 2:-- MS1 Reinigung beenden --, 3: VW_COMMENT
      ;ENDFOLD
      ;FOLD A1864 = AUS ;%{SE}%MKUKATPVW %CVW_SPS %VBOASG %P 2:A1864 = AUS, 3: BOASG
         $OUT[1864] = FALSE
      ;ENDFOLD
      ;FOLD -- MS1 Ausblasen AUS -- ;%{SE}%MKUKATPVW %CVW_COM %VCOMMENT %P 2:-- MS1 Ausblasen AUS --, 3: VW_COMMENT
      ;ENDFOLD
      ;FOLD A1870 = AUS ;%{SE}%MKUKATPVW %CVW_SPS %VBOASG %P 2:A1870 = AUS, 3: BOASG
         $OUT[1870] = FALSE
      ;ENDFOLD
      ;FOLD -- MS1 Einspruehen EIN -- ;%{SE}%MKUKATPVW %CVW_COM %VCOMMENT %P 2:-- MS1 Einspruehen EIN --, 3: VW_COMMENT
      ;ENDFOLD
      ;FOLD A520 = !F574 & F575 ;%{SE}%MKUKATPVW %CVW_SPS %VBOASG %P 2:A520 = !F574 & F575, 3: BOASG
         $OUT[520] = NOT $FLAG[574] AND $FLAG[575]
      ;ENDFOLD
      ;FOLD A1871 = F574 & F575 ;%{SE}%MKUKATPVW %CVW_SPS %VBOASG %P 2:A1871 = F574 & F575, 3: BOASG
         $OUT[1871] = $FLAG[574] AND $FLAG[575]
      ;ENDFOLD
      ;FOLD -- Einschaltdauer Einspruehen -- ;%{SE}%MKUKATPVW %CVW_COM %VCOMMENT %P 2:-- Einschaltdauer Einspruehen --, 3: VW_COMMENT
      ;ENDFOLD
      ;FOLD t7 ( EIN ) = i23[1/10Sek] ;%{SE}%MKUKATPVW %CVW_SPS %VTASG %P 2:t7 ( EIN ) = i23[1/10Sek], 3: TASG
         VW(#SET_TIME,TRUE,7,0,$COUNT_I[23])
      ;ENDFOLD
      ;FOLD Schritt 136 = (F271 + E1864 & !F271) & A4039  ;%{SE}%MKUKATPVW %CVW_SPS %VST_CON %P 2:Schritt 136 = (F271 + E1864 & !F271) & A4039 , 3: ST_CON
         IF ($FLAG[271] OR $IN[1864] AND NOT $FLAG[271]) AND $OUT[4039] THEN
            PREVSTEP = $APP_INT[5]
            $APP_INT[5] = 136
         ENDIF
      ;ENDFOLD
   ;ENDFOLD
   ;FOLD SCHRITT 136 -- MS1 Reinigung (an KS3) -- ;%{P}%MKUKATPVW,%CSTEP,%VST_NR,%P 1:SCHRITT, 2:136, 3: MS1 Reinigung (an KS3)
      ;FOLD ;%{H}
         Case 136
      ;ENDFOLD
      ;FOLD F323 = AUS ;%{SE}%MKUKATPVW %CVW_SPS %VBOASG %P 2:F323 = AUS, 3: BOASG
         $FLAG[323] = FALSE
      ;ENDFOLD
      ;FOLD -- Ueberwachungszeit KS3 schwenken -- ;%{SE}%MKUKATPVW %CVW_COM %VCOMMENT %P 2:-- Ueberwachungszeit KS3 schwenken --, 3: VW_COMMENT
      ;ENDFOLD
      ;FOLD t8 ( EIN ) = -100[1/10Sek] ;%{SE}%MKUKATPVW %CVW_SPS %VTASG %P 2:t8 ( EIN ) = -100[1/10Sek], 3: TASG
         VW(#SET_TIME,TRUE,8,0,-100)
      ;ENDFOLD
      ;FOLD Schritt 137 = T7 & A4039  ;%{SE}%MKUKATPVW %CVW_SPS %VST_CON %P 2:Schritt 137 = T7 & A4039 , 3: ST_CON
         IF $TIMER_FLAG[7] AND $OUT[4039] THEN
            PREVSTEP = $APP_INT[5]
            $APP_INT[5] = 137
         ENDIF
      ;ENDFOLD
   ;ENDFOLD
   ;FOLD SCHRITT 137 -- MS1 Reinigung (an KS3) -- ;%{P}%MKUKATPVW,%CSTEP,%VST_NR,%P 1:SCHRITT, 2:137, 3: MS1 Reinigung (an KS3)
      ;FOLD ;%{H}
         Case 137
      ;ENDFOLD
      ;FOLD -- MS1 Einspruehen AUS -- ;%{SE}%MKUKATPVW %CVW_COM %VCOMMENT %P 2:-- MS1 Einspruehen AUS --, 3: VW_COMMENT
      ;ENDFOLD
      ;FOLD A520 = AUS ;%{SE}%MKUKATPVW %CVW_SPS %VBOASG %P 2:A520 = AUS, 3: BOASG
         $OUT[520] = FALSE
      ;ENDFOLD
      ;FOLD A1871 = AUS ;%{SE}%MKUKATPVW %CVW_SPS %VBOASG %P 2:A1871 = AUS, 3: BOASG
         $OUT[1871] = FALSE
      ;ENDFOLD
      ;FOLD -- RSK Fehlerausgabe KS3 Ruhest. -- ;%{SE}%MKUKATPVW %CVW_COM %VCOMMENT %P 2:-- RSK Fehlerausgabe KS3 Ruhest. --, 3: VW_COMMENT
      ;ENDFOLD
      ;FOLD F324 = !E1163 ;%{SE}%MKUKATPVW %CVW_SPS %VBOASG %P 2:F324 = !E1163, 3: BOASG
         $FLAG[324] = NOT $IN[1163]
      ;ENDFOLD
      ;FOLD -- RSK Sammelstoerung -- ;%{SE}%MKUKATPVW %CVW_COM %VCOMMENT %P 2:-- RSK Sammelstoerung --, 3: VW_COMMENT
      ;ENDFOLD
      ;FOLD F329 = F324 + T8 ;%{SE}%MKUKATPVW %CVW_SPS %VBOASG %P 2:F329 = F324 + T8, 3: BOASG
         $FLAG[329] = $FLAG[324] OR $TIMER_FLAG[8]
      ;ENDFOLD
      ;FOLD Schritt 136 = (E26 + E27) & F324 & A4039  ;%{SE}%MKUKATPVW %CVW_SPS %VST_CON %P 2:Schritt 136 = (E26 + E27) & F324 & A4039 , 3: ST_CON
         IF ($IN[26] OR $IN[27]) AND $FLAG[324] AND $OUT[4039] THEN
            PREVSTEP = $APP_INT[5]
            $APP_INT[5] = 136
         ENDIF
      ;ENDFOLD
      ;FOLD Schritt 138 = (!F324 + T8) & A4039  ;%{SE}%MKUKATPVW %CVW_SPS %VST_CON %P 2:Schritt 138 = (!F324 + T8) & A4039 , 3: ST_CON
         IF (NOT $FLAG[324] OR $TIMER_FLAG[8]) AND $OUT[4039] THEN
            PREVSTEP = $APP_INT[5]
            $APP_INT[5] = 138
         ENDIF
      ;ENDFOLD
   ;ENDFOLD
   ;FOLD SCHRITT 138 -- MS1 Reinigung (an KS3) -- ;%{P}%MKUKATPVW,%CSTEP,%VST_NR,%P 1:SCHRITT, 2:138, 3: MS1 Reinigung (an KS3)
      ;FOLD ;%{H}
         Case 138
      ;ENDFOLD
      ;FOLD -- KS3 in Ruhestellung schwenken -- ;%{SE}%MKUKATPVW %CVW_COM %VCOMMENT %P 2:-- KS3 in Ruhestellung schwenken --, 3: VW_COMMENT
      ;ENDFOLD
      ;FOLD A1162 = !E1162 ;%{SE}%MKUKATPVW %CVW_SPS %VBOASG %P 2:A1162 = !E1162, 3: BOASG
         $OUT[1162] = NOT $IN[1162]
      ;ENDFOLD
      ;FOLD Schritt 139 = A4039  ;%{SE}%MKUKATPVW %CVW_SPS %VST_CON %P 2:Schritt 139 = A4039 , 3: ST_CON
         IF $OUT[4039] THEN
            PREVSTEP = $APP_INT[5]
            $APP_INT[5] = 139
         ENDIF
      ;ENDFOLD
   ;ENDFOLD
   ;FOLD SCHRITT 139 -- MS1 Reinigung (an KS3) -- ;%{P}%MKUKATPVW,%CSTEP,%VST_NR,%P 1:SCHRITT, 2:139, 3: MS1 Reinigung (an KS3)
      ;FOLD ;%{H}
         Case 139
      ;ENDFOLD
      ;FOLD -- RSK Fehlerausgabe KS3 Ruhestellung -- ;%{SE}%MKUKATPVW %CVW_COM %VCOMMENT %P 2:-- RSK Fehlerausgabe KS3 Ruhestellung --, 3: VW_COMMENT
      ;ENDFOLD
      ;FOLD F323 = !E1162 & T8 + F323 ;%{SE}%MKUKATPVW %CVW_SPS %VBOASG %P 2:F323 = !E1162 & T8 + F323, 3: BOASG
         $FLAG[323] = NOT $IN[1162] AND $TIMER_FLAG[8] OR $FLAG[323]
      ;ENDFOLD
      ;FOLD -- RSK Sammelstoerung -- ;%{SE}%MKUKATPVW %CVW_COM %VCOMMENT %P 2:-- RSK Sammelstoerung --, 3: VW_COMMENT
      ;ENDFOLD
      ;FOLD F329 = F323 ;%{SE}%MKUKATPVW %CVW_SPS %VBOASG %P 2:F329 = F323, 3: BOASG
         $FLAG[329] = $FLAG[323]
      ;ENDFOLD
      ;FOLD Schritt 136 = F323 & (E26 + E27) & A4039  ;%{SE}%MKUKATPVW %CVW_SPS %VST_CON %P 2:Schritt 136 = F323 & (E26 + E27) & A4039 , 3: ST_CON
         IF $FLAG[323] AND ($IN[26] OR $IN[27]) AND $OUT[4039] THEN
            PREVSTEP = $APP_INT[5]
            $APP_INT[5] = 136
         ENDIF
      ;ENDFOLD
      ;FOLD Schritt 140 = E1162 & !E1164 & A4039  ;%{SE}%MKUKATPVW %CVW_SPS %VST_CON %P 2:Schritt 140 = E1162 & !E1164 & A4039 , 3: ST_CON
         IF $IN[1162] AND NOT $IN[1164] AND $OUT[4039] THEN
            PREVSTEP = $APP_INT[5]
            $APP_INT[5] = 140
         ENDIF
      ;ENDFOLD
   ;ENDFOLD
   ;FOLD SCHRITT 140 -- MS1 Reinigung (an KS3) -- ;%{P}%MKUKATPVW,%CSTEP,%VST_NR,%P 1:SCHRITT, 2:140, 3: MS1 Reinigung (an KS3)
      ;FOLD ;%{H}
         Case 140
      ;ENDFOLD
      ;FOLD F323 = AUS ;%{SE}%MKUKATPVW %CVW_SPS %VBOASG %P 2:F323 = AUS, 3: BOASG
         $FLAG[323] = FALSE
      ;ENDFOLD
      ;FOLD F329 = AUS ;%{SE}%MKUKATPVW %CVW_SPS %VBOASG %P 2:F329 = AUS, 3: BOASG
         $FLAG[329] = FALSE
      ;ENDFOLD
      ;FOLD -- MS1 Zaehler ruecksetzen -- ;%{SE}%MKUKATPVW %CVW_COM %VCOMMENT %P 2:-- MS1 Zaehler ruecksetzen --, 3: VW_COMMENT
      ;ENDFOLD
      ;FOLD -- MS1 FRG Reinigung -- ;%{SE}%MKUKATPVW %CVW_COM %VCOMMENT %P 2:-- MS1 FRG Reinigung --, 3: VW_COMMENT
      ;ENDFOLD
      ;FOLD F603 = AUS ;%{SE}%MKUKATPVW %CVW_SPS %VBOASG %P 2:F603 = AUS, 3: BOASG
         $FLAG[603] = FALSE
      ;ENDFOLD
      ;FOLD -- MS1 Reinigung FK -- ;%{SE}%MKUKATPVW %CVW_COM %VCOMMENT %P 2:-- MS1 Reinigung FK --, 3: VW_COMMENT
      ;ENDFOLD
      ;FOLD F605 = EIN ;%{SE}%MKUKATPVW %CVW_SPS %VBOASG %P 2:F605 = EIN, 3: BOASG
         $FLAG[605] = TRUE
      ;ENDFOLD
      ;FOLD t8 ( EIN ) = STOP ;%{SE}%MKUKATPVW %CVW_SPS %VTSTOP %P 2:t8 ( EIN ) = STOP, 3: TSTOP
         VW(#SET_TIME,TRUE,8,1,0)
      ;ENDFOLD
      ;FOLD Schritt 1 = A4039  ;%{SE}%MKUKATPVW %CVW_SPS %VST_CON %P 2:Schritt 1 = A4039 , 3: ST_CON
         IF $OUT[4039] THEN
            PREVSTEP = $APP_INT[5]
            $APP_INT[5] = 1
         ENDIF
      ;ENDFOLD
   ;ENDFOLD
   ;FOLD SCHRITT 141 -- MS2 Reinigung (an KS2) -- ;%{P}%MKUKATPVW,%CSTEP,%VST_NR,%P 1:SCHRITT, 2:141, 3: MS2 Reinigung (an KS2)
      ;FOLD ;%{H}
         Case 141
      ;ENDFOLD
      ;FOLD -- RSK gestartet -- ;%{SE}%MKUKATPVW %CVW_COM %VCOMMENT %P 2:-- RSK gestartet --, 3: VW_COMMENT
      ;ENDFOLD
      ;FOLD F321 = AUS ;%{SE}%MKUKATPVW %CVW_SPS %VBOASG %P 2:F321 = AUS, 3: BOASG
         $FLAG[321] = FALSE
      ;ENDFOLD
      ;FOLD F323 = AUS ;%{SE}%MKUKATPVW %CVW_SPS %VBOASG %P 2:F323 = AUS, 3: BOASG
         $FLAG[323] = FALSE
      ;ENDFOLD
      ;FOLD F324 = AUS ;%{SE}%MKUKATPVW %CVW_SPS %VBOASG %P 2:F324 = AUS, 3: BOASG
         $FLAG[324] = FALSE
      ;ENDFOLD
      ;FOLD F329 = AUS ;%{SE}%MKUKATPVW %CVW_SPS %VBOASG %P 2:F329 = AUS, 3: BOASG
         $FLAG[329] = FALSE
      ;ENDFOLD
      ;FOLD -- MS2 Reinigung gestartet -- ;%{SE}%MKUKATPVW %CVW_COM %VCOMMENT %P 2:-- MS2 Reinigung gestartet --, 3: VW_COMMENT
      ;ENDFOLD
      ;FOLD F608 = EIN ;%{SE}%MKUKATPVW %CVW_SPS %VBOASG %P 2:F608 = EIN, 3: BOASG
         $FLAG[608] = TRUE
      ;ENDFOLD
      ;FOLD -- MS bei Reinigung -- ;%{SE}%MKUKATPVW %CVW_COM %VCOMMENT %P 2:-- MS bei Reinigung --, 3: VW_COMMENT
      ;ENDFOLD
      ;FOLD A116 = EIN ;%{SE}%MKUKATPVW %CVW_SPS %VBOASG %P 2:A116 = EIN, 3: BOASG
         $OUT[116] = TRUE
      ;ENDFOLD
      ;FOLD -- Ueberwachungszeit KS2 schwenken -- ;%{SE}%MKUKATPVW %CVW_COM %VCOMMENT %P 2:-- Ueberwachungszeit KS2 schwenken --, 3: VW_COMMENT
      ;ENDFOLD
      ;FOLD t8 ( EIN ) = -50[1/10Sek] ;%{SE}%MKUKATPVW %CVW_SPS %VTASG %P 2:t8 ( EIN ) = -50[1/10Sek], 3: TASG
         VW(#SET_TIME,TRUE,8,0,-50)
      ;ENDFOLD
      ;FOLD Schritt 142 = A4039  ;%{SE}%MKUKATPVW %CVW_SPS %VST_CON %P 2:Schritt 142 = A4039 , 3: ST_CON
         IF $OUT[4039] THEN
            PREVSTEP = $APP_INT[5]
            $APP_INT[5] = 142
         ENDIF
      ;ENDFOLD
   ;ENDFOLD
   ;FOLD SCHRITT 142 -- MS2 Reinigung (an KS2) -- ;%{P}%MKUKATPVW,%CSTEP,%VST_NR,%P 1:SCHRITT, 2:142, 3: MS2 Reinigung (an KS2)
      ;FOLD ;%{H}
         Case 142
      ;ENDFOLD
      ;FOLD -- RSK Fehlerausgabe KS2 Ruhest. -- ;%{SE}%MKUKATPVW %CVW_COM %VCOMMENT %P 2:-- RSK Fehlerausgabe KS2 Ruhest. --, 3: VW_COMMENT
      ;ENDFOLD
      ;FOLD F323 = !E1002 ;%{SE}%MKUKATPVW %CVW_SPS %VBOASG %P 2:F323 = !E1002, 3: BOASG
         $FLAG[323] = NOT $IN[1002]
      ;ENDFOLD
      ;FOLD -- RSK Sammelstoerung -- ;%{SE}%MKUKATPVW %CVW_COM %VCOMMENT %P 2:-- RSK Sammelstoerung --, 3: VW_COMMENT
      ;ENDFOLD
      ;FOLD F329 = F323 ;%{SE}%MKUKATPVW %CVW_SPS %VBOASG %P 2:F329 = F323, 3: BOASG
         $FLAG[329] = $FLAG[323]
      ;ENDFOLD
      ;FOLD Schritt 141 = (E26 + E27) & F323 & A4039  ;%{SE}%MKUKATPVW %CVW_SPS %VST_CON %P 2:Schritt 141 = (E26 + E27) & F323 & A4039 , 3: ST_CON
         IF ($IN[26] OR $IN[27]) AND $FLAG[323] AND $OUT[4039] THEN
            PREVSTEP = $APP_INT[5]
            $APP_INT[5] = 141
         ENDIF
      ;ENDFOLD
      ;FOLD Schritt 143 = (!F323 + T8) & A4039  ;%{SE}%MKUKATPVW %CVW_SPS %VST_CON %P 2:Schritt 143 = (!F323 + T8) & A4039 , 3: ST_CON
         IF (NOT $FLAG[323] OR $TIMER_FLAG[8]) AND $OUT[4039] THEN
            PREVSTEP = $APP_INT[5]
            $APP_INT[5] = 143
         ENDIF
      ;ENDFOLD
   ;ENDFOLD
   ;FOLD SCHRITT 143 -- MS2 Reinigung (an KS2) -- ;%{P}%MKUKATPVW,%CSTEP,%VST_NR,%P 1:SCHRITT, 2:143, 3: MS2 Reinigung (an KS2)
      ;FOLD ;%{H}
         Case 143
      ;ENDFOLD
      ;FOLD -- KS2 in Arbeitsstellung schwenken -- ;%{SE}%MKUKATPVW %CVW_COM %VCOMMENT %P 2:-- KS2 in Arbeitsstellung schwenken --, 3: VW_COMMENT
      ;ENDFOLD
      ;FOLD A1002 = !E1003 ;%{SE}%MKUKATPVW %CVW_SPS %VBOASG %P 2:A1002 = !E1003, 3: BOASG
         $OUT[1002] = NOT $IN[1003]
      ;ENDFOLD
      ;FOLD Schritt 144 = A4039  ;%{SE}%MKUKATPVW %CVW_SPS %VST_CON %P 2:Schritt 144 = A4039 , 3: ST_CON
         IF $OUT[4039] THEN
            PREVSTEP = $APP_INT[5]
            $APP_INT[5] = 144
         ENDIF
      ;ENDFOLD
   ;ENDFOLD
   ;FOLD SCHRITT 144 -- MS2 Reinigung (an KS2) -- ;%{P}%MKUKATPVW,%CSTEP,%VST_NR,%P 1:SCHRITT, 2:144, 3: MS2 Reinigung (an KS2)
      ;FOLD ;%{H}
         Case 144
      ;ENDFOLD
      ;FOLD -- RSK Fehlerausgabe KS2 Arbeitsstellung -- ;%{SE}%MKUKATPVW %CVW_COM %VCOMMENT %P 2:-- RSK Fehlerausgabe KS2 Arbeitsstellung --, 3: VW_COMMENT
      ;ENDFOLD
      ;FOLD F324 = !E1003 & T8 + F324 ;%{SE}%MKUKATPVW %CVW_SPS %VBOASG %P 2:F324 = !E1003 & T8 + F324, 3: BOASG
         $FLAG[324] = NOT $IN[1003] AND $TIMER_FLAG[8] OR $FLAG[324]
      ;ENDFOLD
      ;FOLD -- RSK Sammelstoerung -- ;%{SE}%MKUKATPVW %CVW_COM %VCOMMENT %P 2:-- RSK Sammelstoerung --, 3: VW_COMMENT
      ;ENDFOLD
      ;FOLD F329 = F324 ;%{SE}%MKUKATPVW %CVW_SPS %VBOASG %P 2:F329 = F324, 3: BOASG
         $FLAG[329] = $FLAG[324]
      ;ENDFOLD
      ;FOLD Schritt 141 = F324 & (E26 + E27) & A4039  ;%{SE}%MKUKATPVW %CVW_SPS %VST_CON %P 2:Schritt 141 = F324 & (E26 + E27) & A4039 , 3: ST_CON
         IF $FLAG[324] AND ($IN[26] OR $IN[27]) AND $OUT[4039] THEN
            PREVSTEP = $APP_INT[5]
            $APP_INT[5] = 141
         ENDIF
      ;ENDFOLD
      ;FOLD Schritt 145 = !F324 & E1003 & !E1005 & A4039  ;%{SE}%MKUKATPVW %CVW_SPS %VST_CON %P 2:Schritt 145 = !F324 & E1003 & !E1005 & A4039 , 3: ST_CON
         IF NOT $FLAG[324] AND $IN[1003] AND NOT $IN[1005] AND $OUT[4039] THEN
            PREVSTEP = $APP_INT[5]
            $APP_INT[5] = 145
         ENDIF
      ;ENDFOLD
   ;ENDFOLD
   ;FOLD SCHRITT 145 -- MS2 Reinigung (an KS2) -- ;%{P}%MKUKATPVW,%CSTEP,%VST_NR,%P 1:SCHRITT, 2:145, 3: MS2 Reinigung (an KS2)
      ;FOLD ;%{H}
         Case 145
      ;ENDFOLD
      ;FOLD A1896 = AUS ;%{SE}%MKUKATPVW %CVW_SPS %VBOASG %P 2:A1896 = AUS, 3: BOASG
         $OUT[1896] = FALSE
      ;ENDFOLD
      ;FOLD A2176 = AUS ;%{SE}%MKUKATPVW %CVW_SPS %VBOASG %P 2:A2176 = AUS, 3: BOASG
         $OUT[2176] = FALSE
      ;ENDFOLD
      ;FOLD -- Ueberwachungszeit Versetzeinheit -- ;%{SE}%MKUKATPVW %CVW_COM %VCOMMENT %P 2:-- Ueberwachungszeit Versetzeinheit --, 3: VW_COMMENT
      ;ENDFOLD
      ;FOLD t8 ( EIN ) = -50[1/10Sek] ;%{SE}%MKUKATPVW %CVW_SPS %VTASG %P 2:t8 ( EIN ) = -50[1/10Sek], 3: TASG
         VW(#SET_TIME,TRUE,8,0,-50)
      ;ENDFOLD
      ;FOLD -- Ueberwachungszeit Reinigung -- ;%{SE}%MKUKATPVW %CVW_COM %VCOMMENT %P 2:-- Ueberwachungszeit Reinigung --, 3: VW_COMMENT
      ;ENDFOLD
      ;FOLD t9 ( EIN ) = -80[1/10Sek] ;%{SE}%MKUKATPVW %CVW_SPS %VTASG %P 2:t9 ( EIN ) = -80[1/10Sek], 3: TASG
         VW(#SET_TIME,TRUE,9,0,-80)
      ;ENDFOLD
      ;FOLD Schritt 146 = A4039  ;%{SE}%MKUKATPVW %CVW_SPS %VST_CON %P 2:Schritt 146 = A4039 , 3: ST_CON
         IF $OUT[4039] THEN
            PREVSTEP = $APP_INT[5]
            $APP_INT[5] = 146
         ENDIF
      ;ENDFOLD
   ;ENDFOLD
   ;FOLD SCHRITT 146 -- MS2 Reinigung (an KS2) -- ;%{P}%MKUKATPVW,%CSTEP,%VST_NR,%P 1:SCHRITT, 2:146, 3: MS2 Reinigung (an KS2)
      ;FOLD ;%{H}
         Case 146
      ;ENDFOLD
      ;FOLD -- RSK Fehlerausgabe Versetzeinheit -- ;%{SE}%MKUKATPVW %CVW_COM %VCOMMENT %P 2:-- RSK Fehlerausgabe Versetzeinheit --, 3: VW_COMMENT
      ;ENDFOLD
      ;FOLD F328 = F585 & T8 ;%{SE}%MKUKATPVW %CVW_SPS %VBOASG %P 2:F328 = F585 & T8, 3: BOASG
         $FLAG[328] = $FLAG[585] AND $TIMER_FLAG[8]
      ;ENDFOLD
      ;FOLD -- RSK Sammelstoerung -- ;%{SE}%MKUKATPVW %CVW_COM %VCOMMENT %P 2:-- RSK Sammelstoerung --, 3: VW_COMMENT
      ;ENDFOLD
      ;FOLD F329 = T8 ;%{SE}%MKUKATPVW %CVW_SPS %VBOASG %P 2:F329 = T8, 3: BOASG
         $FLAG[329] = $TIMER_FLAG[8]
      ;ENDFOLD
      ;FOLD F271 = i26 = 0 ;%{SE}%MKUKATPVW %CVW_SPS %VBOCMP %P 2:F271 = i26 = 0, 3: BOCMP
         $FLAG[271] = $COUNT_I[26] == 0
      ;ENDFOLD
      ;FOLD t7 ( F271 ) = -20[1/10Sek] ;%{SE}%MKUKATPVW %CVW_SPS %VTASG %P 2:t7 ( F271 ) = -20[1/10Sek], 3: TASG
         VW(#SET_TIME,$FLAG[271],7,0,-20)
      ;ENDFOLD
      ;FOLD t7 ( !F271 ) = i26[1/10Sek] ;%{SE}%MKUKATPVW %CVW_SPS %VTASG %P 2:t7 ( !F271 ) = i26[1/10Sek], 3: TASG
         VW(#SET_TIME,NOT $FLAG[271],7,0,$COUNT_I[26])
      ;ENDFOLD
      ;FOLD -- Versetzeinheit in Arbeitsst. schw. -- ;%{SE}%MKUKATPVW %CVW_COM %VCOMMENT %P 2:-- Versetzeinheit in Arbeitsst. schw. --, 3: VW_COMMENT
      ;ENDFOLD
      ;FOLD A2176 = !E2176 & F585 ;%{SE}%MKUKATPVW %CVW_SPS %VBOASG %P 2:A2176 = !E2176 & F585, 3: BOASG
         $OUT[2176] = NOT $IN[2176] AND $FLAG[585]
      ;ENDFOLD
      ;FOLD Schritt 145 = A2176 & T8 & (E26 + E27) & A4039  ;%{SE}%MKUKATPVW %CVW_SPS %VST_CON %P 2:Schritt 145 = A2176 & T8 & (E26 + E27) & A4039 , 3: ST_CON
         IF $OUT[2176] AND $TIMER_FLAG[8] AND ($IN[26] OR $IN[27]) AND $OUT[4039] THEN
            PREVSTEP = $APP_INT[5]
            $APP_INT[5] = 145
         ENDIF
      ;ENDFOLD
      ;FOLD Schritt 147 = (E2176 & F585 + !E2168 & !F585) & A4039  ;%{SE}%MKUKATPVW %CVW_SPS %VST_CON %P 2:Schritt 147 = (E2176 & F585 + !E2168 & !F585) & A4039 , 3: ST_CON
         IF ($IN[2176] AND $FLAG[585] OR NOT $IN[2168] AND NOT $FLAG[585]) AND $OUT[4039] THEN
            PREVSTEP = $APP_INT[5]
            $APP_INT[5] = 147
         ENDIF
      ;ENDFOLD
   ;ENDFOLD
   ;FOLD SCHRITT 147 -- MS2 Reinigung (an KS2) -- ;%{P}%MKUKATPVW,%CSTEP,%VST_NR,%P 1:SCHRITT, 2:147, 3: MS2 Reinigung (an KS2)
      ;FOLD ;%{H}
         Case 147
      ;ENDFOLD
      ;FOLD -- RSK Sammelstoerung -- ;%{SE}%MKUKATPVW %CVW_COM %VCOMMENT %P 2:-- RSK Sammelstoerung --, 3: VW_COMMENT
      ;ENDFOLD
      ;FOLD F329 = T9 ;%{SE}%MKUKATPVW %CVW_SPS %VBOASG %P 2:F329 = T9, 3: BOASG
         $FLAG[329] = $TIMER_FLAG[9]
      ;ENDFOLD
      ;FOLD -- MS2 Ausblasen EIN -- ;%{SE}%MKUKATPVW %CVW_COM %VCOMMENT %P 2:-- MS2 Ausblasen EIN --, 3: VW_COMMENT
      ;ENDFOLD
      ;FOLD A1902 = EIN ;%{SE}%MKUKATPVW %CVW_SPS %VBOASG %P 2:A1902 = EIN, 3: BOASG
         $OUT[1902] = TRUE
      ;ENDFOLD
      ;FOLD -- MS2 Reinigung starten -- ;%{SE}%MKUKATPVW %CVW_COM %VCOMMENT %P 2:-- MS2 Reinigung starten --, 3: VW_COMMENT
      ;ENDFOLD
      ;FOLD A1896 = EIN ;%{SE}%MKUKATPVW %CVW_SPS %VBOASG %P 2:A1896 = EIN, 3: BOASG
         $OUT[1896] = TRUE
      ;ENDFOLD
      ;FOLD Schritt 145 = (!E1896 + E1896 & !F271) & T9 & (E26 + E27) & A4039  ;%{SE}%MKUKATPVW %CVW_SPS %VST_CON %P 2:Schritt 145 = (!E1896 + E1896 & !F271) & T9 & (E26 + E27) & A4039 , 3: ST_CON
         IF (NOT $IN[1896] OR $IN[1896] AND NOT $FLAG[271]) AND $TIMER_FLAG[9] AND ($IN[26] OR $IN[27]) AND $OUT[4039] THEN
            PREVSTEP = $APP_INT[5]
            $APP_INT[5] = 145
         ENDIF
      ;ENDFOLD
      ;FOLD Schritt 148 = (E1896 + !E1896 & !F271 & T7) & A4039  ;%{SE}%MKUKATPVW %CVW_SPS %VST_CON %P 2:Schritt 148 = (E1896 + !E1896 & !F271 & T7) & A4039 , 3: ST_CON
         IF ($IN[1896] OR NOT $IN[1896] AND NOT $FLAG[271] AND $TIMER_FLAG[7]) AND $OUT[4039] THEN
            PREVSTEP = $APP_INT[5]
            $APP_INT[5] = 148
         ENDIF
      ;ENDFOLD
   ;ENDFOLD
   ;FOLD SCHRITT 148 -- MS2 Reinigung (an KS2) -- ;%{P}%MKUKATPVW,%CSTEP,%VST_NR,%P 1:SCHRITT, 2:148, 3: MS2 Reinigung (an KS2)
      ;FOLD ;%{H}
         Case 148
      ;ENDFOLD
      ;FOLD -- MS2 Reinigung beenden -- ;%{SE}%MKUKATPVW %CVW_COM %VCOMMENT %P 2:-- MS2 Reinigung beenden --, 3: VW_COMMENT
      ;ENDFOLD
      ;FOLD A1896 = AUS ;%{SE}%MKUKATPVW %CVW_SPS %VBOASG %P 2:A1896 = AUS, 3: BOASG
         $OUT[1896] = FALSE
      ;ENDFOLD
      ;FOLD -- MS2 Ausblasen AUS -- ;%{SE}%MKUKATPVW %CVW_COM %VCOMMENT %P 2:-- MS2 Ausblasen AUS --, 3: VW_COMMENT
      ;ENDFOLD
      ;FOLD A1902 = AUS ;%{SE}%MKUKATPVW %CVW_SPS %VBOASG %P 2:A1902 = AUS, 3: BOASG
         $OUT[1902] = FALSE
      ;ENDFOLD
      ;FOLD -- MS2 Einspruehen EIN -- ;%{SE}%MKUKATPVW %CVW_COM %VCOMMENT %P 2:-- MS2 Einspruehen EIN --, 3: VW_COMMENT
      ;ENDFOLD
      ;FOLD A528 = !F583 & F584 ;%{SE}%MKUKATPVW %CVW_SPS %VBOASG %P 2:A528 = !F583 & F584, 3: BOASG
         $OUT[528] = NOT $FLAG[583] AND $FLAG[584]
      ;ENDFOLD
      ;FOLD A1903 = F583 & F584 ;%{SE}%MKUKATPVW %CVW_SPS %VBOASG %P 2:A1903 = F583 & F584, 3: BOASG
         $OUT[1903] = $FLAG[583] AND $FLAG[584]
      ;ENDFOLD
      ;FOLD -- Einschaltdauer Einspruehen -- ;%{SE}%MKUKATPVW %CVW_COM %VCOMMENT %P 2:-- Einschaltdauer Einspruehen --, 3: VW_COMMENT
      ;ENDFOLD
      ;FOLD t7 ( EIN ) = i23[1/10Sek] ;%{SE}%MKUKATPVW %CVW_SPS %VTASG %P 2:t7 ( EIN ) = i23[1/10Sek], 3: TASG
         VW(#SET_TIME,TRUE,7,0,$COUNT_I[23])
      ;ENDFOLD
      ;FOLD Schritt 149 = (F271 + E1896 & !F271) & A4039  ;%{SE}%MKUKATPVW %CVW_SPS %VST_CON %P 2:Schritt 149 = (F271 + E1896 & !F271) & A4039 , 3: ST_CON
         IF ($FLAG[271] OR $IN[1896] AND NOT $FLAG[271]) AND $OUT[4039] THEN
            PREVSTEP = $APP_INT[5]
            $APP_INT[5] = 149
         ENDIF
      ;ENDFOLD
   ;ENDFOLD
   ;FOLD SCHRITT 149 -- MS2 Reinigung (an KS2) -- ;%{P}%MKUKATPVW,%CSTEP,%VST_NR,%P 1:SCHRITT, 2:149, 3: MS2 Reinigung (an KS2)
      ;FOLD ;%{H}
         Case 149
      ;ENDFOLD
      ;FOLD F323 = AUS ;%{SE}%MKUKATPVW %CVW_SPS %VBOASG %P 2:F323 = AUS, 3: BOASG
         $FLAG[323] = FALSE
      ;ENDFOLD
      ;FOLD -- Ueberwachungszeit KS2 schwenken -- ;%{SE}%MKUKATPVW %CVW_COM %VCOMMENT %P 2:-- Ueberwachungszeit KS2 schwenken --, 3: VW_COMMENT
      ;ENDFOLD
      ;FOLD t8 ( EIN ) = -100[1/10Sek] ;%{SE}%MKUKATPVW %CVW_SPS %VTASG %P 2:t8 ( EIN ) = -100[1/10Sek], 3: TASG
         VW(#SET_TIME,TRUE,8,0,-100)
      ;ENDFOLD
      ;FOLD Schritt 150 = T7 & A4039  ;%{SE}%MKUKATPVW %CVW_SPS %VST_CON %P 2:Schritt 150 = T7 & A4039 , 3: ST_CON
         IF $TIMER_FLAG[7] AND $OUT[4039] THEN
            PREVSTEP = $APP_INT[5]
            $APP_INT[5] = 150
         ENDIF
      ;ENDFOLD
   ;ENDFOLD
   ;FOLD SCHRITT 150 -- MS2 Reinigung (an KS2) -- ;%{P}%MKUKATPVW,%CSTEP,%VST_NR,%P 1:SCHRITT, 2:150, 3: MS2 Reinigung (an KS2)
      ;FOLD ;%{H}
         Case 150
      ;ENDFOLD
      ;FOLD -- MS2 Einspruehen AUS -- ;%{SE}%MKUKATPVW %CVW_COM %VCOMMENT %P 2:-- MS2 Einspruehen AUS --, 3: VW_COMMENT
      ;ENDFOLD
      ;FOLD A528 = AUS ;%{SE}%MKUKATPVW %CVW_SPS %VBOASG %P 2:A528 = AUS, 3: BOASG
         $OUT[528] = FALSE
      ;ENDFOLD
      ;FOLD A1903 = AUS ;%{SE}%MKUKATPVW %CVW_SPS %VBOASG %P 2:A1903 = AUS, 3: BOASG
         $OUT[1903] = FALSE
      ;ENDFOLD
      ;FOLD -- RSK Fehlerausgabe KS2 Ruhest. -- ;%{SE}%MKUKATPVW %CVW_COM %VCOMMENT %P 2:-- RSK Fehlerausgabe KS2 Ruhest. --, 3: VW_COMMENT
      ;ENDFOLD
      ;FOLD F324 = !E1003 ;%{SE}%MKUKATPVW %CVW_SPS %VBOASG %P 2:F324 = !E1003, 3: BOASG
         $FLAG[324] = NOT $IN[1003]
      ;ENDFOLD
      ;FOLD -- RSK Sammelstoerung -- ;%{SE}%MKUKATPVW %CVW_COM %VCOMMENT %P 2:-- RSK Sammelstoerung --, 3: VW_COMMENT
      ;ENDFOLD
      ;FOLD F329 = F324 ;%{SE}%MKUKATPVW %CVW_SPS %VBOASG %P 2:F329 = F324, 3: BOASG
         $FLAG[329] = $FLAG[324]
      ;ENDFOLD
      ;FOLD Schritt 149 = (E26 + E27) & F324 & A4039  ;%{SE}%MKUKATPVW %CVW_SPS %VST_CON %P 2:Schritt 149 = (E26 + E27) & F324 & A4039 , 3: ST_CON
         IF ($IN[26] OR $IN[27]) AND $FLAG[324] AND $OUT[4039] THEN
            PREVSTEP = $APP_INT[5]
            $APP_INT[5] = 149
         ENDIF
      ;ENDFOLD
      ;FOLD Schritt 151 = (!F324 + T8) & A4039  ;%{SE}%MKUKATPVW %CVW_SPS %VST_CON %P 2:Schritt 151 = (!F324 + T8) & A4039 , 3: ST_CON
         IF (NOT $FLAG[324] OR $TIMER_FLAG[8]) AND $OUT[4039] THEN
            PREVSTEP = $APP_INT[5]
            $APP_INT[5] = 151
         ENDIF
      ;ENDFOLD
   ;ENDFOLD
   ;FOLD SCHRITT 151 -- MS2 Reinigung (an KS2) -- ;%{P}%MKUKATPVW,%CSTEP,%VST_NR,%P 1:SCHRITT, 2:151, 3: MS2 Reinigung (an KS2)
      ;FOLD ;%{H}
         Case 151
      ;ENDFOLD
      ;FOLD -- KS2 in Ruhestellung schwenken -- ;%{SE}%MKUKATPVW %CVW_COM %VCOMMENT %P 2:-- KS2 in Ruhestellung schwenken --, 3: VW_COMMENT
      ;ENDFOLD
      ;FOLD A1002 = !E1002 ;%{SE}%MKUKATPVW %CVW_SPS %VBOASG %P 2:A1002 = !E1002, 3: BOASG
         $OUT[1002] = NOT $IN[1002]
      ;ENDFOLD
      ;FOLD Schritt 152 = A4039  ;%{SE}%MKUKATPVW %CVW_SPS %VST_CON %P 2:Schritt 152 = A4039 , 3: ST_CON
         IF $OUT[4039] THEN
            PREVSTEP = $APP_INT[5]
            $APP_INT[5] = 152
         ENDIF
      ;ENDFOLD
   ;ENDFOLD
   ;FOLD SCHRITT 152 -- MS2 Reinigung (an KS2) -- ;%{P}%MKUKATPVW,%CSTEP,%VST_NR,%P 1:SCHRITT, 2:152, 3: MS2 Reinigung (an KS2)
      ;FOLD ;%{H}
         Case 152
      ;ENDFOLD
      ;FOLD -- RSK Fehlerausgabe KS2 Ruhestellung -- ;%{SE}%MKUKATPVW %CVW_COM %VCOMMENT %P 2:-- RSK Fehlerausgabe KS2 Ruhestellung --, 3: VW_COMMENT
      ;ENDFOLD
      ;FOLD F323 = !E1002 & T8 + F323 ;%{SE}%MKUKATPVW %CVW_SPS %VBOASG %P 2:F323 = !E1002 & T8 + F323, 3: BOASG
         $FLAG[323] = NOT $IN[1002] AND $TIMER_FLAG[8] OR $FLAG[323]
      ;ENDFOLD
      ;FOLD -- RSK Sammelstoerung -- ;%{SE}%MKUKATPVW %CVW_COM %VCOMMENT %P 2:-- RSK Sammelstoerung --, 3: VW_COMMENT
      ;ENDFOLD
      ;FOLD F329 = F323 ;%{SE}%MKUKATPVW %CVW_SPS %VBOASG %P 2:F329 = F323, 3: BOASG
         $FLAG[329] = $FLAG[323]
      ;ENDFOLD
      ;FOLD Schritt 149 = F323 & (E26 + E27) & A4039  ;%{SE}%MKUKATPVW %CVW_SPS %VST_CON %P 2:Schritt 149 = F323 & (E26 + E27) & A4039 , 3: ST_CON
         IF $FLAG[323] AND ($IN[26] OR $IN[27]) AND $OUT[4039] THEN
            PREVSTEP = $APP_INT[5]
            $APP_INT[5] = 149
         ENDIF
      ;ENDFOLD
      ;FOLD Schritt 153 = E1002 & !E1004 & A4039  ;%{SE}%MKUKATPVW %CVW_SPS %VST_CON %P 2:Schritt 153 = E1002 & !E1004 & A4039 , 3: ST_CON
         IF $IN[1002] AND NOT $IN[1004] AND $OUT[4039] THEN
            PREVSTEP = $APP_INT[5]
            $APP_INT[5] = 153
         ENDIF
      ;ENDFOLD
   ;ENDFOLD
   ;FOLD SCHRITT 153 -- MS2 Reinigung (an KS2) -- ;%{P}%MKUKATPVW,%CSTEP,%VST_NR,%P 1:SCHRITT, 2:153, 3: MS2 Reinigung (an KS2)
      ;FOLD ;%{H}
         Case 153
      ;ENDFOLD
      ;FOLD F323 = AUS ;%{SE}%MKUKATPVW %CVW_SPS %VBOASG %P 2:F323 = AUS, 3: BOASG
         $FLAG[323] = FALSE
      ;ENDFOLD
      ;FOLD F329 = AUS ;%{SE}%MKUKATPVW %CVW_SPS %VBOASG %P 2:F329 = AUS, 3: BOASG
         $FLAG[329] = FALSE
      ;ENDFOLD
      ;FOLD -- MS2 Zaehler ruecksetzen -- ;%{SE}%MKUKATPVW %CVW_COM %VCOMMENT %P 2:-- MS2 Zaehler ruecksetzen --, 3: VW_COMMENT
      ;ENDFOLD
      ;FOLD -- MS2 FRG Reinigung -- ;%{SE}%MKUKATPVW %CVW_COM %VCOMMENT %P 2:-- MS2 FRG Reinigung --, 3: VW_COMMENT
      ;ENDFOLD
      ;FOLD F607 = AUS ;%{SE}%MKUKATPVW %CVW_SPS %VBOASG %P 2:F607 = AUS, 3: BOASG
         $FLAG[607] = FALSE
      ;ENDFOLD
      ;FOLD -- MS2 Reinigung FK -- ;%{SE}%MKUKATPVW %CVW_COM %VCOMMENT %P 2:-- MS2 Reinigung FK --, 3: VW_COMMENT
      ;ENDFOLD
      ;FOLD F609 = EIN ;%{SE}%MKUKATPVW %CVW_SPS %VBOASG %P 2:F609 = EIN, 3: BOASG
         $FLAG[609] = TRUE
      ;ENDFOLD
      ;FOLD t8 ( EIN ) = STOP ;%{SE}%MKUKATPVW %CVW_SPS %VTSTOP %P 2:t8 ( EIN ) = STOP, 3: TSTOP
         VW(#SET_TIME,TRUE,8,1,0)
      ;ENDFOLD
      ;FOLD Schritt 1 = A4039  ;%{SE}%MKUKATPVW %CVW_SPS %VST_CON %P 2:Schritt 1 = A4039 , 3: ST_CON
         IF $OUT[4039] THEN
            PREVSTEP = $APP_INT[5]
            $APP_INT[5] = 1
         ENDIF
      ;ENDFOLD
   ;ENDFOLD
   ;FOLD SCHRITT 154 -- MS1 Reinigung (an Pneum. Schwenkeinheit MS1)-- ;%{P}%MKUKATPVW,%CSTEP,%VST_NR,%P 1:SCHRITT, 2:154, 3: MS1 Reinigung (an Pneum. Schwenkeinheit MS1)
      ;FOLD ;%{H}
         Case 154
      ;ENDFOLD
      ;FOLD -- RSK gestartet -- ;%{SE}%MKUKATPVW %CVW_COM %VCOMMENT %P 2:-- RSK gestartet --, 3: VW_COMMENT
      ;ENDFOLD
      ;FOLD F321 = AUS ;%{SE}%MKUKATPVW %CVW_SPS %VBOASG %P 2:F321 = AUS, 3: BOASG
         $FLAG[321] = FALSE
      ;ENDFOLD
      ;FOLD F323 = AUS ;%{SE}%MKUKATPVW %CVW_SPS %VBOASG %P 2:F323 = AUS, 3: BOASG
         $FLAG[323] = FALSE
      ;ENDFOLD
      ;FOLD F324 = AUS ;%{SE}%MKUKATPVW %CVW_SPS %VBOASG %P 2:F324 = AUS, 3: BOASG
         $FLAG[324] = FALSE
      ;ENDFOLD
      ;FOLD F329 = AUS ;%{SE}%MKUKATPVW %CVW_SPS %VBOASG %P 2:F329 = AUS, 3: BOASG
         $FLAG[329] = FALSE
      ;ENDFOLD
      ;FOLD -- MS1 Reinigung gestartet -- ;%{SE}%MKUKATPVW %CVW_COM %VCOMMENT %P 2:-- MS1 Reinigung gestartet --, 3: VW_COMMENT
      ;ENDFOLD
      ;FOLD F604 = EIN ;%{SE}%MKUKATPVW %CVW_SPS %VBOASG %P 2:F604 = EIN, 3: BOASG
         $FLAG[604] = TRUE
      ;ENDFOLD
      ;FOLD -- MS bei Reinigung -- ;%{SE}%MKUKATPVW %CVW_COM %VCOMMENT %P 2:-- MS bei Reinigung --, 3: VW_COMMENT
      ;ENDFOLD
      ;FOLD A116 = EIN ;%{SE}%MKUKATPVW %CVW_SPS %VBOASG %P 2:A116 = EIN, 3: BOASG
         $OUT[116] = TRUE
      ;ENDFOLD
      ;FOLD -- Steuerluft EIN -- ;%{SE}%MKUKATPVW %CVW_COM %VCOMMENT %P 2:-- Steuerluft EIN --, 3: VW_COMMENT
      ;ENDFOLD
      ;FOLD A2161 = A4039 ;%{SE}%MKUKATPVW %CVW_SPS %VBOASG %P 2:A2161 = A4039, 3: BOASG
         $OUT[2161] = $OUT[4039]
      ;ENDFOLD
      ;FOLD A2163 = AUS ;%{SE}%MKUKATPVW %CVW_SPS %VBOASG %P 2:A2163 = AUS, 3: BOASG
         $OUT[2163] = FALSE
      ;ENDFOLD
      ;FOLD A2164 = AUS ;%{SE}%MKUKATPVW %CVW_SPS %VBOASG %P 2:A2164 = AUS, 3: BOASG
         $OUT[2164] = FALSE
      ;ENDFOLD
      ;FOLD A2165 = AUS ;%{SE}%MKUKATPVW %CVW_SPS %VBOASG %P 2:A2165 = AUS, 3: BOASG
         $OUT[2165] = FALSE
      ;ENDFOLD
      ;FOLD A2166 = AUS ;%{SE}%MKUKATPVW %CVW_SPS %VBOASG %P 2:A2166 = AUS, 3: BOASG
         $OUT[2166] = FALSE
      ;ENDFOLD
      ;FOLD A2167 = AUS ;%{SE}%MKUKATPVW %CVW_SPS %VBOASG %P 2:A2167 = AUS, 3: BOASG
         $OUT[2167] = FALSE
      ;ENDFOLD
      ;FOLD A2168 = AUS ;%{SE}%MKUKATPVW %CVW_SPS %VBOASG %P 2:A2168 = AUS, 3: BOASG
         $OUT[2168] = FALSE
      ;ENDFOLD
      ;FOLD -- Ueberwachungszeit Schwenkeinheit 1 -- ;%{SE}%MKUKATPVW %CVW_COM %VCOMMENT %P 2:-- Ueberwachungszeit Schwenkeinheit 1 --, 3: VW_COMMENT
      ;ENDFOLD
      ;FOLD t8 ( EIN ) = -100[1/10Sek] ;%{SE}%MKUKATPVW %CVW_SPS %VTASG %P 2:t8 ( EIN ) = -100[1/10Sek], 3: TASG
         VW(#SET_TIME,TRUE,8,0,-100)
      ;ENDFOLD
      ;FOLD Schritt 155 = A4039  ;%{SE}%MKUKATPVW %CVW_SPS %VST_CON %P 2:Schritt 155 = A4039 , 3: ST_CON
         IF $OUT[4039] THEN
            PREVSTEP = $APP_INT[5]
            $APP_INT[5] = 155
         ENDIF
      ;ENDFOLD
   ;ENDFOLD
   ;FOLD SCHRITT 155 -- MS1 Reinigung (an Pneum. Schwenkeinheit MS1)-- ;%{P}%MKUKATPVW,%CSTEP,%VST_NR,%P 1:SCHRITT, 2:155, 3: MS1 Reinigung (an Pneum. Schwenkeinheit MS1)
      ;FOLD ;%{H}
         Case 155
      ;ENDFOLD
      ;FOLD -- Steuerluft EIN -- ;%{SE}%MKUKATPVW %CVW_COM %VCOMMENT %P 2:-- Steuerluft EIN --, 3: VW_COMMENT
      ;ENDFOLD
      ;FOLD A2161 = A4039 ;%{SE}%MKUKATPVW %CVW_SPS %VBOASG %P 2:A2161 = A4039, 3: BOASG
         $OUT[2161] = $OUT[4039]
      ;ENDFOLD
      ;FOLD -- RSK Fehlerausgabe Schwenkeinheit 1 Ruhest. -- ;%{SE}%MKUKATPVW %CVW_COM %VCOMMENT %P 2:-- RSK Fehlerausgabe Schwenkeinheit 1 Ruhest. --, 3: VW_COMMENT
      ;ENDFOLD
      ;FOLD F323 = !E2163 & T8 ;%{SE}%MKUKATPVW %CVW_SPS %VBOASG %P 2:F323 = !E2163 & T8, 3: BOASG
         $FLAG[323] = NOT $IN[2163] AND $TIMER_FLAG[8]
      ;ENDFOLD
      ;FOLD -- RSK Sammelstoerung -- ;%{SE}%MKUKATPVW %CVW_COM %VCOMMENT %P 2:-- RSK Sammelstoerung --, 3: VW_COMMENT
      ;ENDFOLD
      ;FOLD F329 = F323 + T8 ;%{SE}%MKUKATPVW %CVW_SPS %VBOASG %P 2:F329 = F323 + T8, 3: BOASG
         $FLAG[329] = $FLAG[323] OR $TIMER_FLAG[8]
      ;ENDFOLD
      ;FOLD Schritt 154 = (E26 + E27) & F323 & A4039  ;%{SE}%MKUKATPVW %CVW_SPS %VST_CON %P 2:Schritt 154 = (E26 + E27) & F323 & A4039 , 3: ST_CON
         IF ($IN[26] OR $IN[27]) AND $FLAG[323] AND $OUT[4039] THEN
            PREVSTEP = $APP_INT[5]
            $APP_INT[5] = 154
         ENDIF
      ;ENDFOLD
      ;FOLD Schritt 156 = (!F323 + T8) & (F523 & !F524 & E2161 + !F523 & F524 & !E2162) & A4039  ;%{SE}%MKUKATPVW %CVW_SPS %VST_CON %P 2:Schritt 156 = (!F323 + T8) & (F523 & !F524 & E2161 + !F523 & F524 & !E2162) & A4039 , 3: ST_CON
         IF (NOT $FLAG[323] OR $TIMER_FLAG[8]) AND ($FLAG[523] AND NOT $FLAG[524] AND $IN[2161] OR NOT $FLAG[523] AND $FLAG[524] AND NOT $IN[2162]) AND $OUT[4039] THEN
            PREVSTEP = $APP_INT[5]
            $APP_INT[5] = 156
         ENDIF
      ;ENDFOLD
   ;ENDFOLD
   ;FOLD SCHRITT 156 -- MS1 Reinigung (an Pneum. Schwenkeinheit MS1)-- ;%{P}%MKUKATPVW,%CSTEP,%VST_NR,%P 1:SCHRITT, 2:156, 3: MS1 Reinigung (an Pneum. Schwenkeinheit MS1)
      ;FOLD ;%{H}
         Case 156
      ;ENDFOLD
      ;FOLD -- Steuerluft EIN -- ;%{SE}%MKUKATPVW %CVW_COM %VCOMMENT %P 2:-- Steuerluft EIN --, 3: VW_COMMENT
      ;ENDFOLD
      ;FOLD A2161 = A4039 ;%{SE}%MKUKATPVW %CVW_SPS %VBOASG %P 2:A2161 = A4039, 3: BOASG
         $OUT[2161] = $OUT[4039]
      ;ENDFOLD
      ;FOLD -- Schwenkeinheit 1 in Arbeitsstellung schwenken -- ;%{SE}%MKUKATPVW %CVW_COM %VCOMMENT %P 2:-- Schwenkeinheit 1 in Arbeitsstellung schwenken --, 3: VW_COMMENT
      ;ENDFOLD
      ;FOLD A2163 = AUS ;%{SE}%MKUKATPVW %CVW_SPS %VBOASG %P 2:A2163 = AUS, 3: BOASG
         $OUT[2163] = FALSE
      ;ENDFOLD
      ;FOLD A2164 = EIN ;%{SE}%MKUKATPVW %CVW_SPS %VBOASG %P 2:A2164 = EIN, 3: BOASG
         $OUT[2164] = TRUE
      ;ENDFOLD
      ;FOLD -- FRG Bewegung EIN -- ;%{SE}%MKUKATPVW %CVW_COM %VCOMMENT %P 2:-- FRG Bewegung EIN --, 3: VW_COMMENT
      ;ENDFOLD
      ;FOLD A2165 = AUS ;%{SE}%MKUKATPVW %CVW_SPS %VBOASG %P 2:A2165 = AUS, 3: BOASG
         $OUT[2165] = FALSE
      ;ENDFOLD
      ;FOLD A2166 = EIN ;%{SE}%MKUKATPVW %CVW_SPS %VBOASG %P 2:A2166 = EIN, 3: BOASG
         $OUT[2166] = TRUE
      ;ENDFOLD
      ;FOLD -- Zeit Endlage entprellen -- ;%{SE}%MKUKATPVW %CVW_COM %VCOMMENT %P 2:-- Zeit Endlage entprellen --, 3: VW_COMMENT
      ;ENDFOLD
      ;FOLD t9 ( !E2164 ) = -10[1/10Sek] ;%{SE}%MKUKATPVW %CVW_SPS %VTASG %P 2:t9 ( !E2164 ) = -10[1/10Sek], 3: TASG
         VW(#SET_TIME,NOT $IN[2164],9,0,-10)
      ;ENDFOLD
      ;FOLD Schritt 157 = E2164 & !E2163 & A4039 & T9 + T8  ;%{SE}%MKUKATPVW %CVW_SPS %VST_CON %P 2:Schritt 157 = E2164 & !E2163 & A4039 & T9 + T8 , 3: ST_CON
         IF $IN[2164] AND NOT $IN[2163] AND $OUT[4039] AND $TIMER_FLAG[9] OR $TIMER_FLAG[8] THEN
            PREVSTEP = $APP_INT[5]
            $APP_INT[5] = 157
         ENDIF
      ;ENDFOLD
   ;ENDFOLD
   ;FOLD SCHRITT 157 -- MS1 Reinigung (an Pneum. Schwenkeinheit MS1)-- ;%{P}%MKUKATPVW,%CSTEP,%VST_NR,%P 1:SCHRITT, 2:157, 3: MS1 Reinigung (an Pneum. Schwenkeinheit MS1)
      ;FOLD ;%{H}
         Case 157
      ;ENDFOLD
      ;FOLD -- Steuerluft EIN -- ;%{SE}%MKUKATPVW %CVW_COM %VCOMMENT %P 2:-- Steuerluft EIN --, 3: VW_COMMENT
      ;ENDFOLD
      ;FOLD A2161 = A4039 ;%{SE}%MKUKATPVW %CVW_SPS %VBOASG %P 2:A2161 = A4039, 3: BOASG
         $OUT[2161] = $OUT[4039]
      ;ENDFOLD
      ;FOLD -- RSK Fehlerausgabe Schwenkeinheit 1 Arbeitsstellung -- ;%{SE}%MKUKATPVW %CVW_COM %VCOMMENT %P 2:-- RSK Fehlerausgabe Schwenkeinheit 1 Arbeitsstellung --, 3: VW_COMMENT
      ;ENDFOLD
